  MoveL 4003 to (327.57, -9.53, -317.09) mm, rotated rx -179.9 ry 0 rz -90 deg; joints [33.762, -56.151, 91.428, -130.036, 46.527, 141.521]
  MoveL 4004 to (328.02, -9.53, -316.88) mm, rotated rx -179.9 ry 0 rz -90 deg; joints [33.78, -56.147, 91.421, -130.014, 46.536, 141.505]
  MoveL 4005 to (328.06, -9.53, -316.86) mm, rotated rx -179.9 ry 0 rz -90 deg; joints [33.782, -56.146, 91.42, -130.012, 46.537, 141.503]
  MoveL 4006 to (328.49, -9.53, -316.61) mm, rotated rx -179.9 ry 0 rz -90 deg; joints [33.8, -56.144, 91.417, -129.992, 46.547, 141.489]
  MoveL 4007 to (328.92, -9.53, -316.31) mm, rotated rx -179.9 ry 0 rz -90 deg; joints [33.819, -56.145, 91.417, -129.971, 46.559, 141.475]
  MoveL 4008 to (329.14, -9.53, -316.14) mm, rotated rx -179.9 ry 0 rz -90 deg; joints [33.829, -56.146, 91.419, -129.961, 46.565, 141.468]
  MoveL 4009 to (329.35, -9.52, -315.96) mm, rotated rx -179.9 ry 0 rz -90 deg; joints [33.839, -56.148, 91.422, -129.951, 46.573, 141.462]
  MoveL 4010 to (329.58, -9.52, -315.74) mm, rotated rx -179.9 ry 0 rz -90 deg; joints [33.85, -56.152, 91.427, -129.94, 46.581, 141.456]
  MoveL 4011 to (329.82, -9.52, -315.49) mm, rotated rx -179.9 ry 0 rz -90 deg; joints [33.862, -56.157, 91.435, -129.929, 46.59, 141.45]
  MoveL 4012 to (330, -9.53, -315.27) mm, rotated rx -179.9 ry 0 rz -90 deg; joints [33.872, -56.161, 91.442, -129.92, 46.598, 141.445]
  MoveL 4013 to (330.17, -9.53, -315.06) mm, rotated rx -179.9 ry 0 rz -90 deg; joints [33.882, -56.167, 91.45, -129.912, 46.606, 141.442]
  MoveL 4014 to (330.47, -9.52, -314.63) mm, rotated rx -179.9 ry 0 rz -90 deg; joints [33.9, -56.178, 91.469, -129.898, 46.621, 141.436]
  MoveL 4015 to (330.72, -9.52, -314.2) mm, rotated rx -179.9 ry 0 rz -90 deg; joints [33.916, -56.192, 91.491, -129.886, 46.636, 141.433]
  MoveL 4016 to (330.74, -9.53, -314.16) mm, rotated rx -179.9 ry 0 rz -90 deg; joints [33.917, -56.193, 91.493, -129.885, 46.638, 141.433]
  MoveL 4017 to (330.95, -9.53, -313.71) mm, rotated rx -179.9 ry 0 rz -90 deg; joints [33.933, -56.209, 91.518, -129.876, 46.654, 141.431]
  MoveL 4018 to (331.12, -9.53, -313.26) mm, rotated rx -179.9 ry 0 rz -90 deg; joints [33.947, -56.227, 91.546, -129.868, 46.669, 141.432]
  MoveL 4019 to (331.26, -9.52, -312.81) mm, rotated rx -179.9 ry 0 rz -90 deg; joints [33.96, -56.245, 91.575, -129.862, 46.685, 141.434]
  MoveL 4020 to (331.35, -9.52, -312.37) mm, rotated rx -179.9 ry 0 rz -90 deg; joints [33.972, -56.265, 91.607, -129.857, 46.7, 141.438]
  MoveL 4021 to (331.42, -9.53, -311.92) mm, rotated rx -179.9 ry 0 rz -90 deg; joints [33.983, -56.286, 91.64, -129.854, 46.715, 141.443]
  MoveL 4022 to (331.45, -9.52, -311.47) mm, rotated rx -179.9 ry 0 rz -90 deg; joints [33.993, -56.308, 91.675, -129.853, 46.729, 141.45]
  MoveL 4023 to (331.45, -9.53, -310.57) mm, rotated rx -179.9 ry 0 rz -90 deg; joints [34.012, -56.354, 91.749, -129.853, 46.759, 141.466]
  MoveL 4024 to (331.45, -9.52, -3.46) mm, rotated rx -179.9 ry 0 rz -90 deg; joints [41.448, -70.91, 113.437, -126.774, 55.713, 144.028]
  MoveL 4025 to (331.45, -9.53, -2.56) mm, rotated rx -179.9 ry 0 rz -90 deg; joints [41.474, -70.95, 113.491, -126.757, 55.737, 144.029]
  MoveL 4026 to (331.42, -9.53, -2.11) mm, rotated rx -179.9 ry 0 rz -90 deg; joints [41.486, -70.971, 113.52, -126.75, 55.749, 144.03]
  MoveL 4027 to (331.36, -9.52, -1.67) mm, rotated rx -179.9 ry 0 rz -90 deg; joints [41.497, -70.993, 113.551, -126.744, 55.76, 144.032]
  MoveL 4028 to (331.27, -9.52, -1.22) mm, rotated rx -179.9 ry 0 rz -90 deg; joints [41.506, -71.016, 113.583, -126.739, 55.771, 144.035]
  MoveL 4029 to (331.14, -9.53, -0.77) mm, rotated rx -179.9 ry 0 rz -90 deg; joints [41.515, -71.041, 113.617, -126.735, 55.782, 144.04]
  MoveL 4030 to (330.97, -9.53, -0.32) mm, rotated rx -179.9 ry 0 rz -90 deg; joints [41.523, -71.068, 113.653, -126.733, 55.792, 144.045]
  MoveL 4031 to (330.77, -9.52, 0.13) mm, rotated rx -179.9 ry 0 rz -90 deg; joints [41.529, -71.096, 113.691, -126.733, 55.802, 144.052]
  MoveL 4032 to (330.72, -9.52, 0.23) mm, rotated rx -179.9 ry 0 rz -90 deg; joints [41.53, -71.102, 113.7, -126.733, 55.804, 144.054]
  MoveL 4033 to (330.49, -9.52, 0.63) mm, rotated rx -179.9 ry 0 rz -90 deg; joints [41.534, -71.128, 113.736, -126.735, 55.812, 144.061]
  MoveL 4034 to (330.21, -9.52, 1.03) mm, rotated rx -179.9 ry 0 rz -90 deg; joints [41.537, -71.157, 113.775, -126.738, 55.82, 144.07]
  MoveL 4035 to (330.03, -9.53, 1.27) mm, rotated rx -179.9 ry 0 rz -90 deg; joints [41.538, -71.175, 113.8, -126.74, 55.825, 144.076]
  MoveL 4036 to (329.82, -9.53, 1.51) mm, rotated rx -179.9 ry 0 rz -90 deg; joints [41.538, -71.193, 113.826, -126.744, 55.829, 144.083]
  MoveL 4037 to (329.62, -9.53, 1.72) mm, rotated rx -179.9 ry 0 rz -90 deg; joints [41.537, -71.21, 113.849, -126.748, 55.833, 144.089]
  MoveL 4038 to (329.41, -9.53, 1.93) mm, rotated rx -179.9 ry 0 rz -90 deg; joints [41.536, -71.228, 113.873, -126.752, 55.836, 144.096]
  MoveL 4039 to (329.16, -9.53, 2.14) mm, rotated rx -179.9 ry 0 rz -90 deg; joints [41.535, -71.247, 113.899, -126.758, 55.839, 144.104]
  MoveL 4040 to (328.92, -9.53, 2.33) mm, rotated rx -179.9 ry 0 rz -90 deg; joints [41.532, -71.265, 113.924, -126.764, 55.842, 144.112]
  MoveL 4041 to (328.54, -9.52, 2.6) mm, rotated rx -179.9 ry 0 rz -90 deg; joints [41.528, -71.291, 113.961, -126.774, 55.845, 144.124]
  MoveL 4042 to (328.16, -9.53, 2.82) mm, rotated rx -179.9 ry 0 rz -90 deg; joints [41.522, -71.316, 113.995, -126.785, 55.847, 144.136]
  MoveL 4043 to (328.02, -9.52, 2.9) mm, rotated rx -179.9 ry 0 rz -90 deg; joints [41.519, -71.324, 114.007, -126.789, 55.848, 144.141]
  MoveL 4044 to (327.57, -9.53, 3.11) mm, rotated rx -179.9 ry 0 rz -90 deg; joints [41.511, -71.351, 114.044, -126.803, 55.849, 144.155]
  MoveL 4045 to (327.12, -9.53, 3.28) mm, rotated rx -179.9 ry 0 rz -90 deg; joints [41.501, -71.376, 114.078, -126.817, 55.849, 144.17]
  MoveL 4046 to (326.67, -9.52, 3.41) mm, rotated rx -179.9 ry 0 rz -90 deg; joints [41.491, -71.399, 114.11, -126.833, 55.848, 144.184]
  MoveL 4047 to (326.22, -9.53, 3.51) mm, rotated rx -179.9 ry 0 rz -90 deg; joints [41.479, -71.421, 114.14, -126.849, 55.846, 144.198]
  MoveL 4048 to (325.77, -9.53, 3.57) mm, rotated rx -179.9 ry 0 rz -90 deg; joints [41.466, -71.441, 114.168, -126.866, 55.844, 144.213]
  MoveL 4049 to (325.33, -9.53, 3.6) mm, rotated rx -179.9 ry 0 rz -90 deg; joints [41.452, -71.46, 114.195, -126.883, 55.84, 144.227]
  MoveL 4050 to (324.43, -9.52, 3.61) mm, rotated rx -179.9 ry 0 rz -90 deg; joints [41.423, -71.495, 114.243, -126.919, 55.831, 144.256]
  MoveL 4051 to (319.96, -9.52, 3.61) mm, rotated rx -179.9 ry 0 rz -90 deg; joints [41.278, -71.667, 114.483, -127.098, 55.786, 144.399]
  MoveL 4052 to (319.95, -9.53, 3.61) mm, rotated rx -179.9 ry 0 rz -90 deg; joints [41.278, -71.668, 114.484, -127.098, 55.786, 144.399]
  MoveL 4053 to (319.93, -9.53, 3.62) mm, rotated rx -179.9 ry 0 rz -90 deg; joints [41.277, -71.669, 114.485, -127.099, 55.787, 144.399]
  MoveL 4054 to (319.83, -9.53, 3.72) mm, rotated rx -179.9 ry 0 rz -90 deg; joints [41.277, -71.678, 114.497, -127.101, 55.788, 144.403]
  MoveL 4055 to (319.43, -9.53, 4.05) mm, rotated rx -179.9 ry 0 rz -90 deg; joints [41.273, -71.707, 114.538, -127.11, 55.793, 144.415]
  MoveL 4056 to (319.03, -9.52, 4.33) mm, rotated rx -179.9 ry 0 rz -90 deg; joints [41.268, -71.735, 114.576, -127.121, 55.796, 144.428]
  MoveL 4057 to (318.78, -9.53, 4.48) mm, rotated rx -179.9 ry 0 rz -90 deg; joints [41.265, -71.751, 114.599, -127.128, 55.798, 144.436]
  MoveL 4058 to (318.54, -9.52, 4.62) mm, rotated rx -179.9 ry 0 rz -90 deg; joints [41.26, -71.767, 114.62, -127.135, 55.799, 144.444]
  MoveL 4059 to (318.14, -9.52, 4.81) mm, rotated rx -179.9 ry 0 rz -90 deg; joints [41.253, -71.791, 114.653, -127.147, 55.8, 144.456]
  MoveL 4060 to (317.69, -9.53, 4.99) mm, rotated rx -179.9 ry 0 rz -90 deg; joints [41.243, -71.816, 114.688, -127.162, 55.8, 144.471]
  MoveL 4061 to (317.24, -9.53, 5.13) mm, rotated rx -179.9 ry 0 rz -90 deg; joints [41.233, -71.84, 114.72, -127.177, 55.799, 144.485]
  MoveL 4062 to (316.79, -9.53, 5.23) mm, rotated rx -179.9 ry 0 rz -90 deg; joints [41.221, -71.862, 114.751, -127.193, 55.797, 144.499]
  MoveL 4063 to (316.34, -9.53, 5.3) mm, rotated rx -179.9 ry 0 rz -90 deg; joints [41.208, -71.882, 114.779, -127.21, 55.795, 144.514]
  MoveL 4064 to (315.89, -9.52, 5.34) mm, rotated rx -179.9 ry 0 rz -90 deg; joints [41.195, -71.901, 114.805, -127.227, 55.791, 144.528]
  MoveL 4065 to (315.44, -9.52, 5.35) mm, rotated rx -179.9 ry 0 rz -90 deg; joints [41.18, -71.919, 114.829, -127.245, 55.787, 144.542]
  MoveL 4066 to (-302.86, -9.53, 5.35) mm, rotated rx -179.9 ry 0 rz -90 deg; joints [14.008, -90.074, 136.69, -160.776, 47.297, 167.14]
  MoveL 4067 to (-303.31, -9.52, 5.35) mm, rotated rx -179.9 ry 0 rz -90 deg; joints [13.983, -90.081, 136.697, -160.809, 47.292, 167.161]
  MoveL 4068 to (-303.76, -9.52, 5.31) mm, rotated rx -179.9 ry 0 rz -90 deg; joints [13.958, -90.086, 136.702, -160.842, 47.286, 167.183]
  MoveL 4069 to (-304.21, -9.53, 5.25) mm, rotated rx -179.9 ry 0 rz -90 deg; joints [13.933, -90.089, 136.705, -160.876, 47.281, 167.206]
  MoveL 4070 to (-304.66, -9.53, 5.15) mm, rotated rx -179.9 ry 0 rz -90 deg; joints [13.907, -90.09, 136.706, -160.91, 47.275, 167.229]
  MoveL 4071 to (-305.1, -9.53, 5.01) mm, rotated rx -179.9 ry 0 rz -90 deg; joints [13.881, -90.088, 136.705, -160.945, 47.269, 167.253]
  MoveL 4072 to (-305.55, -9.52, 4.84) mm, rotated rx -179.9 ry 0 rz -90 deg; joints [13.854, -90.084, 136.701, -160.981, 47.264, 167.276]
  MoveL 4073 to (-306.02, -9.52, 4.62) mm, rotated rx -179.9 ry 0 rz -90 deg; joints [13.825, -90.077, 136.695, -161.019, 47.258, 167.302]
  MoveL 4074 to (-306.45, -9.53, 4.37) mm, rotated rx -179.9 ry 0 rz -90 deg; joints [13.798, -90.067, 136.685, -161.055, 47.252, 167.326]
  MoveL 4075 to (-306.88, -9.53, 4.07) mm, rotated rx -179.9 ry 0 rz -90 deg; joints [13.771, -90.054, 136.673, -161.092, 47.247, 167.35]
  MoveL 4076 to (-307.31, -9.52, 3.72) mm, rotated rx -179.9 ry 0 rz -90 deg; joints [13.743, -90.038, 136.657, -161.129, 47.241, 167.376]
  MoveL 4077 to (-307.35, -9.53, 3.68) mm, rotated rx -179.9 ry 0 rz -90 deg; joints [13.74, -90.036, 136.656, -161.133, 47.241, 167.378]
  MoveL 4078 to (-307.41, -9.53, 3.63) mm, rotated rx -179.9 ry 0 rz -90 deg; joints [13.736, -90.033, 136.653, -161.138, 47.24, 167.382]
  MoveL 4079 to (-307.42, -9.53, 3.62) mm, rotated rx -179.9 ry 0 rz -90 deg; joints [13.735, -90.033, 136.652, -161.139, 47.24, 167.382]
  MoveL 4080 to (-307.44, -9.53, 3.61) mm, rotated rx -179.9 ry 0 rz -90 deg; joints [13.734, -90.032, 136.652, -161.141, 47.239, 167.383]
  MoveL 4081 to (-319.03, -9.53, 3.61) mm, rotated rx -179.9 ry 0 rz -90 deg; joints [13.099, -90.213, 136.836, -161.987, 47.104, 167.949]
  MoveL 4082 to (-319.93, -9.52, 3.6) mm, rotated rx -179.9 ry 0 rz -90 deg; joints [13.049, -90.226, 136.849, -162.053, 47.094, 167.993]
  MoveL 4083 to (-320.38, -9.52, 3.56) mm, rotated rx -179.9 ry 0 rz -90 deg; joints [13.024, -90.23, 136.854, -162.087, 47.089, 168.016]
  MoveL 4084 to (-320.83, -9.52, 3.48) mm, rotated rx -179.9 ry 0 rz -90 deg; joints [12.998, -90.232, 136.856, -162.121, 47.084, 168.039]
  MoveL 4085 to (-321.28, -9.53, 3.38) mm, rotated rx -179.9 ry 0 rz -90 deg; joints [12.972, -90.232, 136.856, -162.156, 47.079, 168.062]
  MoveL 4086 to (-321.73, -9.53, 3.24) mm, rotated rx -179.9 ry 0 rz -90 deg; joints [12.946, -90.229, 136.854, -162.192, 47.073, 168.086]
  MoveL 4087 to (-321.8, -9.53, 3.21) mm, rotated rx -179.9 ry 0 rz -90 deg; joints [12.941, -90.229, 136.853, -162.197, 47.072, 168.09]
  MoveC 4088 to (-322.89, -9.52, 3.37) mm, rotated rx -179.9 ry 0 rz -90 deg; joints [12.883, -90.256, 136.88, -162.275, 47.06, 168.142] to (-323.45, -9.52, 4.32) mm, rotated rx -179.9 ry 0 rz -90 deg; joints [12.865, -90.327, 136.95, -162.299, 47.055, 168.158]
  MoveL 4089 to (-323.45, -9.52, 4.32) mm, rotated rx -179.9 ry 0 rz -90 deg; joints [12.865, -90.327, 136.95, -162.299, 47.055, 168.158]
  MoveL 4090 to (-323.82, -9.52, 8.63) mm, rotated rx -179.9 ry 0 rz -90 deg; joints [12.899, -90.621, 137.235, -162.25, 47.054, 168.123]
  MoveL 4091 to (-323.89, -9.15, 9.52) mm, rotated rx -179.9 ry 0 rz -90 deg; joints [12.907, -90.7, 137.28, -162.231, 47.022, 168.103]
  MoveL 4092 to (-323.92, -8.26, 9.89) mm, rotated rx -179.9 ry 0 rz -90 deg; joints [12.909, -90.77, 137.271, -162.205, 46.948, 168.067]
  Set speed (1000.0 mm/s)
  MoveL 4093 to (-323.92, 25.52, 9.89) mm, rotated rx -179.9 ry 0 rz -90 deg; joints [12.895, -92.363, 135.971, -161.337, 44.198, 166.814]
  Print: /'90 deg cut'
  Call SetTool(1)
  Set speed (1000.0 mm/s)
  MoveL 4094 to (-315.62, 25.53, -1.4) mm, rotated rx -179.9 ry 0 rz -90 deg; joints [13.207, -91.468, 135.125, -160.92, 44.317, 166.531]
  MoveL 4095 to (-315.62, 12.75, -1.4) mm, rotated rx -179.9 ry 0 rz -90 deg; joints [13.212, -90.888, 135.622, -161.264, 45.337, 167.021]
  Set speed (100.0 mm/s)
  MoveL 4096 to (-315.62, 5.79, -1.4) mm, rotated rx -179.9 ry 0 rz -90 deg; joints [13.215, -90.564, 135.888, -161.444, 45.896, 167.282]
  MoveC 4097 to (-315.25, 4.9, -1.4) mm, rotated rx -179.9 ry 0 rz -90 deg; joints [13.235, -90.516, 135.916, -161.44, 45.973, 167.296] to (-314.35, 4.53, -1.4) mm, rotated rx -179.9 ry 0 rz -90 deg; joints [13.284, -90.484, 135.916, -161.383, 46.014, 167.265]
  MoveL 4098 to (-314.35, 4.53, -1.4) mm, rotated rx -179.9 ry 0 rz -90 deg; joints [13.284, -90.484, 135.916, -161.383, 46.014, 167.265]
  MoveL 4099 to (-310.68, 4.52, -1.4) mm, rotated rx -179.9 ry 0 rz -90 deg; joints [13.485, -90.427, 135.858, -161.112, 46.058, 167.08]
  MoveC 4100 to (-309.78, 4.52, -1.77) mm, rotated rx -179.9 ry 0 rz -90 deg; joints [13.529, -90.388, 135.819, -161.052, 46.069, 167.04] to (-309.41, 4.53, -2.67) mm, rotated rx -179.9 ry 0 rz -90 deg; joints [13.537, -90.322, 135.755, -161.042, 46.072, 167.033]
  MoveL 4101 to (-309.41, 4.53, -2.67) mm, rotated rx -179.9 ry 0 rz -90 deg; joints [13.537, -90.322, 135.755, -161.042, 46.072, 167.033]
  MoveL 4102 to (-309.41, 4.52, -311.19) mm, rotated rx -179.9 ry 0 rz -90 deg; joints [10.394, -71.426, 113.61, -164.457, 42.297, 168.759]
  MoveL 4103 to (-309.41, 4.53, -311.26) mm, rotated rx -179.9 ry 0 rz -90 deg; joints [10.393, -71.421, 113.604, -164.458, 42.296, 168.759]
  MoveL 4104 to (-309.41, 4.52, -311.3) mm, rotated rx -179.9 ry 0 rz -90 deg; joints [10.393, -71.419, 113.601, -164.458, 42.295, 168.759]
  MoveL 4105 to (-309.41, 4.52, -311.32) mm, rotated rx -179.9 ry 0 rz -90 deg; joints [10.393, -71.418, 113.6, -164.458, 42.295, 168.759]
  MoveC 4106 to (-309.88, 4.52, -312.32) mm, rotated rx -179.9 ry 0 rz -90 deg; joints [10.365, -71.365, 113.527, -164.493, 42.271, 168.781] to (-310.96, 4.53, -312.57) mm, rotated rx -179.9 ry 0 rz -90 deg; joints [10.317, -71.361, 113.523, -164.562, 42.261, 168.831]
  MoveL 4107 to (-310.96, 4.52, -312.57) mm, rotated rx -179.9 ry 0 rz -90 deg; joints [10.317, -71.361, 113.523, -164.562, 42.261, 168.831]
  MoveL 4108 to (-314.37, 4.53, -311.79) mm, rotated rx -179.9 ry 0 rz -90 deg; joints [10.178, -71.442, 113.635, -164.774, 42.263, 168.991]
  MoveL 4109 to (-315.24, 4.9, -311.59) mm, rotated rx -179.9 ry 0 rz -90 deg; joints [10.143, -71.476, 113.652, -164.821, 42.24, 169.022]
  MoveL 4110 to (-315.61, 5.79, -311.51) mm, rotated rx -179.9 ry 0 rz -90 deg; joints [10.128, -71.517, 113.635, -164.826, 42.182, 169.016]
  Set speed (1000.0 mm/s)
  MoveL 4111 to (-315.61, 15.52, -311.51) mm, rotated rx -179.9 ry 0 rz -90 deg; joints [10.125, -71.863, 113.325, -164.637, 41.548, 168.76]
  MoveL 4112 to (-316.42, 15.53, -1.4) mm, rotated rx -179.9 ry 0 rz -90 deg; joints [13.167, -91.028, 135.528, -161.25, 45.105, 166.957]
  MoveL 4113 to (-316.42, 7, -1.4) mm, rotated rx -179.9 ry 0 rz -90 deg; joints [13.171, -90.632, 135.854, -161.472, 45.79, 167.277]
  Set speed (100.0 mm/s)
  MoveL 4114 to (-316.42, 1.27, -1.4) mm, rotated rx -179.9 ry 0 rz -90 deg; joints [13.173, -90.362, 136.07, -161.618, 46.252, 167.489]
  MoveC 4115 to (-316.05, 0.37, -1.4) mm, rotated rx -179.9 ry 0 rz -90 deg; joints [13.194, -90.313, 136.098, -161.613, 46.329, 167.504] to (-315.15, 0, -1.4) mm, rotated rx -179.9 ry 0 rz -90 deg; joints [13.243, -90.282, 136.098, -161.556, 46.369, 167.472]
  MoveL 4116 to (-315.15, 0, -1.4) mm, rotated rx -179.9 ry 0 rz -90 deg; joints [13.243, -90.282, 136.098, -161.556, 46.369, 167.472]
  MoveL 4117 to (-310.68, 0, -1.4) mm, rotated rx -179.9 ry 0 rz -90 deg; joints [13.487, -90.212, 136.028, -161.228, 46.423, 167.25]
  MoveC 4118 to (-309.78, 0, -1.77) mm, rotated rx -179.9 ry 0 rz -90 deg; joints [13.531, -90.173, 135.989, -161.169, 46.433, 167.21] to (-309.41, 0, -2.67) mm, rotated rx -179.9 ry 0 rz -90 deg; joints [13.539, -90.108, 135.925, -161.158, 46.436, 167.203]
  MoveL 4119 to (-309.41, 0, -2.67) mm, rotated rx -179.9 ry 0 rz -90 deg; joints [13.539, -90.108, 135.925, -161.158, 46.436, 167.203]
  MoveL 4120 to (-309.41, 0, -311.19) mm, rotated rx -179.9 ry 0 rz -90 deg; joints [10.395, -71.262, 113.751, -164.544, 42.592, 168.878]
  MoveL 4121 to (-309.41, 0, -311.26) mm, rotated rx -179.9 ry 0 rz -90 deg; joints [10.395, -71.258, 113.745, -164.545, 42.59, 168.878]
  MoveL 4122 to (-309.41, 0, -311.3) mm, rotated rx -179.9 ry 0 rz -90 deg; joints [10.394, -71.255, 113.742, -164.545, 42.589, 168.878]
  MoveL 4123 to (-309.41, 0, -311.32) mm, rotated rx -179.9 ry 0 rz -90 deg; joints [10.394, -71.254, 113.741, -164.545, 42.589, 168.878]
  MoveC 4124 to (-309.88, 0, -312.31) mm, rotated rx -179.9 ry 0 rz -90 deg; joints [10.367, -71.201, 113.669, -164.579, 42.565, 168.899] to (-310.95, 0, -312.57) mm, rotated rx -179.9 ry 0 rz -90 deg; joints [10.319, -71.197, 113.664, -164.648, 42.555, 168.949]
  MoveL 4125 to (-310.95, 0, -312.57) mm, rotated rx -179.9 ry 0 rz -90 deg; joints [10.319, -71.197, 113.664, -164.648, 42.555, 168.949]
  MoveL 4126 to (-315.17, 0, -311.67) mm, rotated rx -179.9 ry 0 rz -90 deg; joints [10.146, -71.294, 113.798, -164.909, 42.558, 169.145]
  MoveL 4127 to (-316.05, 0.37, -311.48) mm, rotated rx -179.9 ry 0 rz -90 deg; joints [10.11, -71.327, 113.814, -164.957, 42.534, 169.176]
  MoveL 4128 to (-316.41, 1.27, -311.4) mm, rotated rx -179.9 ry 0 rz -90 deg; joints [10.095, -71.368, 113.797, -164.962, 42.476, 169.17]
  Set speed (1000.0 mm/s)
  MoveL 4129 to (-316.41, 16.53, -311.4) mm, rotated rx -179.9 ry 0 rz -90 deg; joints [10.091, -71.913, 113.313, -164.669, 41.481, 168.772]
  MoveL 4130 to (328.05, 16.53, -312.66) mm, rotated rx -179.9 ry 0 rz -90 deg; joints [33.855, -57.084, 90.962, -128.897, 45.696, 139.954]
  MoveL 4131 to (328.05, 12.76, -312.66) mm, rotated rx -179.9 ry 0 rz -90 deg; joints [33.857, -56.983, 91.082, -129.063, 45.837, 140.193]
  Set speed (100.0 mm/s)
  MoveL 4132 to (328.05, 5.79, -312.66) mm, rotated rx -179.9 ry 0 rz -90 deg; joints [33.86, -56.792, 91.301, -129.366, 46.098, 140.632]
  MoveL 4133 to (327.68, 4.9, -312.65) mm, rotated rx -179.9 ry 0 rz -90 deg; joints [33.849, -56.781, 91.35, -129.423, 46.129, 140.705]
  MoveL 4134 to (326.78, 4.53, -312.64) mm, rotated rx -179.9 ry 0 rz -90 deg; joints [33.823, -56.802, 91.413, -129.482, 46.139, 140.769]
  MoveL 4135 to (323.18, 4.53, -312.6) mm, rotated rx -179.9 ry 0 rz -90 deg; joints [33.714, -56.928, 91.617, -129.656, 46.12, 140.931]
  MoveC 4136 to (322.29, 4.52, -312.22) mm, rotated rx -179.9 ry 0 rz -90 deg; joints [33.695, -56.978, 91.698, -129.7, 46.127, 140.978] to (321.93, 4.52, -311.32) mm, rotated rx -179.9 ry 0 rz -90 deg; joints [33.702, -57.038, 91.793, -129.718, 46.154, 141.011]
  MoveL 4137 to (321.93, 4.52, -311.32) mm, rotated rx -179.9 ry 0 rz -90 deg; joints [33.702, -57.038, 91.793, -129.718, 46.154, 141.011]
  MoveL 4138 to (321.93, 4.52, -311.3) mm, rotated rx -179.9 ry 0 rz -90 deg; joints [33.703, -57.039, 91.794, -129.718, 46.155, 141.011]
  MoveL 4139 to (321.93, 4.53, -311.26) mm, rotated rx -179.9 ry 0 rz -90 deg; joints [33.703, -57.041, 91.797, -129.718, 46.156, 141.012]
  MoveL 4140 to (321.93, 4.53, -311.04) mm, rotated rx -179.9 ry 0 rz -90 deg; joints [33.708, -57.052, 91.815, -129.718, 46.163, 141.015]
  MoveL 4141 to (321.93, 4.52, -2.67) mm, rotated rx -179.9 ry 0 rz -90 deg; joints [41.154, -71.823, 113.563, -126.625, 55.068, 143.42]
  MoveC 4142 to (322.41, 4.53, -1.67) mm, rotated rx -179.9 ry 0 rz -90 deg; joints [41.198, -71.849, 113.597, -126.587, 55.099, 143.404] to (323.5, 4.53, -1.43) mm, rotated rx -179.9 ry 0 rz -90 deg; joints [41.24, -71.818, 113.553, -126.539, 55.117, 143.369]
  MoveL 4143 to (323.5, 4.52, -1.43) mm, rotated rx -179.9 ry 0 rz -90 deg; joints [41.24, -71.818, 113.553, -126.539, 55.117, 143.369]
  MoveL 4144 to (326.89, 4.53, -2.25) mm, rotated rx -179.9 ry 0 rz -90 deg; joints [41.327, -71.649, 113.322, -126.419, 55.131, 143.26]
  MoveL 4145 to (327.76, 4.9, -2.46) mm, rotated rx -179.9 ry 0 rz -90 deg; joints [41.349, -71.619, 113.25, -126.374, 55.12, 143.207]
  MoveL 4146 to (328.13, 5.8, -2.54) mm, rotated rx -179.9 ry 0 rz -90 deg; joints [41.358, -71.633, 113.197, -126.328, 55.086, 143.137]
  Set speed (1000.0 mm/s)
  MoveL 4147 to (328.13, 15.52, -2.54) mm, rotated rx -179.9 ry 0 rz -90 deg; joints [41.352, -71.977, 112.885, -125.962, 54.696, 142.493]
  MoveL 4148 to (328.88, 15.52, -312.67) mm, rotated rx -179.9 ry 0 rz -90 deg; joints [33.881, -57.028, 90.947, -128.901, 45.738, 139.98]
  MoveL 4149 to (328.88, 7, -312.67) mm, rotated rx -179.9 ry 0 rz -90 deg; joints [33.884, -56.796, 91.216, -129.274, 46.057, 140.519]
  Set speed (100.0 mm/s)
  MoveL 4150 to (328.88, 1.27, -312.67) mm, rotated rx -179.9 ry 0 rz -90 deg; joints [33.887, -56.638, 91.394, -129.52, 46.272, 140.877]
  MoveL 4151 to (328.51, 0.37, -312.66) mm, rotated rx -179.9 ry 0 rz -90 deg; joints [33.876, -56.626, 91.442, -129.577, 46.303, 140.95]
  MoveL 4152 to (327.61, 0, -312.65) mm, rotated rx -179.9 ry 0 rz -90 deg; joints [33.849, -56.647, 91.505, -129.636, 46.313, 141.013]
  MoveL 4153 to (323.18, 0, -312.6) mm, rotated rx -179.9 ry 0 rz -90 deg; joints [33.716, -56.802, 91.756, -129.85, 46.291, 141.213]
  MoveC 4154 to (322.29, 0, -312.22) mm, rotated rx -179.9 ry 0 rz -90 deg; joints [33.697, -56.852, 91.838, -129.893, 46.298, 141.259] to (321.93, 0, -311.32) mm, rotated rx -179.9 ry 0 rz -90 deg; joints [33.704, -56.911, 91.932, -129.911, 46.326, 141.292]
  MoveL 4155 to (321.93, 0, -311.32) mm, rotated rx -179.9 ry 0 rz -90 deg; joints [33.704, -56.911, 91.932, -129.911, 46.326, 141.292]
  MoveL 4156 to (321.93, 0, -311.3) mm, rotated rx -179.9 ry 0 rz -90 deg; joints [33.705, -56.912, 91.934, -129.911, 46.326, 141.292]
  MoveL 4157 to (321.93, 0, -311.26) mm, rotated rx -179.9 ry 0 rz -90 deg; joints [33.705, -56.914, 91.937, -129.911, 46.328, 141.293]
  MoveL 4158 to (321.93, 0, -311.04) mm, rotated rx -179.9 ry 0 rz -90 deg; joints [33.71, -56.926, 91.955, -129.911, 46.335, 141.296]
  MoveL 4159 to (321.93, 0, -2.67) mm, rotated rx -179.9 ry 0 rz -90 deg; joints [41.157, -71.66, 113.705, -126.793, 55.252, 143.716]
  MoveC 4160 to (322.41, 0, -1.67) mm, rotated rx -179.9 ry 0 rz -90 deg; joints [41.201, -71.686, 113.739, -126.755, 55.283, 143.701] to (323.48, 0, -1.43) mm, rotated rx -179.9 ry 0 rz -90 deg; joints [41.243, -71.656, 113.697, -126.707, 55.3, 143.666]
  MoveL 4161 to (323.48, 0, -1.43) mm, rotated rx -179.9 ry 0 rz -90 deg; joints [41.243, -71.656, 113.697, -126.707, 55.3, 143.666]
  MoveL 4162 to (327.69, 0, -2.38) mm, rotated rx -179.9 ry 0 rz -90 deg; joints [41.352, -71.45, 113.412, -126.557, 55.319, 143.531]
  MoveL 4163 to (328.57, 0.37, -2.58) mm, rotated rx -179.9 ry 0 rz -90 deg; joints [41.375, -71.42, 113.341, -126.512, 55.308, 143.478]
  MoveL 4164 to (328.93, 1.27, -2.66) mm, rotated rx -179.9 ry 0 rz -90 deg; joints [41.383, -71.435, 113.289, -126.466, 55.273, 143.407]
  Set speed (1000.0 mm/s)
  MoveL 4165 to (328.93, 25.52, -2.66) mm, rotated rx -179.9 ry 0 rz -90 deg; joints [41.369, -72.285, 112.507, -125.548, 54.305, 141.799]
  Print: /'diagnonal cut'
  Call SetTool(1)
  Set speed (1000.0 mm/s)
  MoveL 4166 to (-336.73, -13.8, 1.64) mm, rotated rx -179.15 ry 0 rz -30.08 deg; joints [-4.609, -80.567, 143.565, -185.552, 62.915, 242.65]
  MoveL 4167 to (-334.14, -15.3, 1.64) mm, rotated rx -179.15 ry 0 rz -30.08 deg; joints [-4.459, -80.469, 143.61, -185.378, 63.051, 242.56]
  Set speed (100.0 mm/s)
  MoveL 4168 to (-328.11, -18.79, 1.64) mm, rotated rx -179.15 ry 0 rz -30.08 deg; joints [-4.111, -80.238, 143.712, -184.973, 63.369, 242.351]
  MoveL 4169 to (-327.17, -18.95, 1.47) mm, rotated rx -179.15 ry 0 rz -30.08 deg; joints [-4.056, -80.22, 143.708, -184.91, 63.38, 242.323]
  MoveL 4170 to (-326.45, -18.45, 1.07) mm, rotated rx -179.15 ry 0 rz -30.08 deg; joints [-4.013, -80.238, 143.672, -184.864, 63.326, 242.306]
  MoveL 4171 to (-325.38, -16.61, 0) mm, rotated rx -179.15 ry 0 rz -30.08 deg; joints [-3.947, -80.317, 143.564, -184.799, 63.137, 242.291]
  MoveC 4172 to (-325.07, -16.06, -0.74) mm, rotated rx -179.15 ry 0 rz -30.08 deg; joints [-3.926, -80.317, 143.502, -184.778, 63.074, 242.286] to (-325.1, -16.12, -1.71) mm, rotated rx -179.15 ry 0 rz -30.08 deg; joints [-3.925, -80.257, 143.435, -184.777, 63.066, 242.286]
  MoveL 4173 to (-325.1, -16.12, -1.71) mm, rotated rx -179.15 ry 0 rz -30.08 deg; joints [-3.925, -80.257, 143.435, -184.777, 63.066, 242.286]
  MoveL 4174 to (-325.19, -16.27, -2.08) mm, rotated rx -179.15 ry 0 rz -30.08 deg; joints [-3.928, -80.225, 143.41, -184.78, 63.074, 242.287]
  MoveL 4175 to (-325.26, -16.39, -2.46) mm, rotated rx -179.15 ry 0 rz -30.08 deg; joints [-3.931, -80.194, 143.386, -184.783, 63.08, 242.288]
  MoveL 4176 to (-325.32, -16.51, -2.91) mm, rotated rx -179.15 ry 0 rz -30.08 deg; joints [-3.933, -80.16, 143.356, -184.785, 63.085, 242.289]
  MoveL 4177 to (-325.37, -16.59, -3.36) mm, rotated rx -179.15 ry 0 rz -30.08 deg; joints [-3.934, -80.128, 143.325, -184.786, 63.086, 242.289]
  MoveL 4178 to (-325.4, -16.65, -3.81) mm, rotated rx -179.15 ry 0 rz -30.08 deg; joints [-3.934, -80.099, 143.294, -184.786, 63.085, 242.289]
  MoveL 4179 to (-325.42, -16.68, -4.26) mm, rotated rx -179.15 ry 0 rz -30.08 deg; joints [-3.933, -80.071, 143.263, -184.785, 63.081, 242.289]
  MoveL 4180 to (-325.42, -16.68, -5.16) mm, rotated rx -179.15 ry 0 rz -30.08 deg; joints [-3.93, -80.02, 143.199, -184.782, 63.068, 242.289]
  MoveL 4181 to (-325.42, -16.68, -310.67) mm, rotated rx -179.15 ry 0 rz -30.08 deg; joints [-3.03, -64.015, 119.968, -184.065, 55.829, 242.408]
  MoveL 4182 to (-325.42, -16.67, -311.57) mm, rotated rx -179.15 ry 0 rz -30.08 deg; joints [-3.028, -63.969, 119.894, -184.064, 55.801, 242.409]
  MoveL 4183 to (-325.4, -16.64, -312.02) mm, rotated rx -179.15 ry 0 rz -30.08 deg; joints [-3.026, -63.949, 119.857, -184.063, 55.784, 242.409]
  MoveL 4184 to (-325.36, -16.57, -312.47) mm, rotated rx -179.15 ry 0 rz -30.08 deg; joints [-3.023, -63.929, 119.82, -184.06, 55.766, 242.408]
  MoveL 4185 to (-325.31, -16.48, -312.92) mm, rotated rx -179.15 ry 0 rz -30.08 deg; joints [-3.02, -63.911, 119.782, -184.057, 55.746, 242.408]
  MoveL 4186 to (-325.24, -16.36, -313.37) mm, rotated rx -179.15 ry 0 rz -30.08 deg; joints [-3.016, -63.895, 119.744, -184.053, 55.724, 242.407]
  MoveL 4187 to (-325.17, -16.25, -313.69) mm, rotated rx -179.15 ry 0 rz -30.08 deg; joints [-3.012, -63.884, 119.716, -184.05, 55.707, 242.406]
  MoveL 4188 to (-325.1, -16.12, -314.02) mm, rotated rx -179.15 ry 0 rz -30.08 deg; joints [-3.008, -63.874, 119.688, -184.046, 55.688, 242.405]
  MoveL 4189 to (-325.04, -16.01, -314.27) mm, rotated rx -179.15 ry 0 rz -30.08 deg; joints [-3.005, -63.867, 119.666, -184.043, 55.673, 242.404]
  MoveL 4190 to (-324.9, -15.78, -314.72) mm, rotated rx -179.15 ry 0 rz -30.08 deg; joints [-2.998, -63.857, 119.626, -184.036, 55.644, 242.402]
  MoveL 4191 to (-324.74, -15.5, -315.17) mm, rotated rx -179.15 ry 0 rz -30.08 deg; joints [-2.99, -63.848, 119.585, -184.028, 55.611, 242.399]
  MoveL 4192 to (-324.65, -15.35, -315.38) mm, rotated rx -179.15 ry 0 rz -30.08 deg; joints [-2.986, -63.845, 119.566, -184.023, 55.595, 242.398]
  MoveL 4193 to (-324.48, -15.05, -315.75) mm, rotated rx -179.15 ry 0 rz -30.08 deg; joints [-2.977, -63.842, 119.532, -184.015, 55.563, 242.394]
  MoveL 4194 to (-324.31, -14.75, -316.07) mm, rotated rx -179.15 ry 0 rz -30.08 deg; joints [-2.969, -63.842, 119.502, -184.006, 55.534, 242.391]
  MoveL 4195 to (-324.2, -14.57, -316.24) mm, rotated rx -179.15 ry 0 rz -30.08 deg; joints [-2.964, -63.842, 119.485, -184.001, 55.517, 242.389]
  MoveL 4196 to (-323.97, -14.18, -316.56) mm, rotated rx -179.15 ry 0 rz -30.08 deg; joints [-2.954, -63.846, 119.454, -183.99, 55.481, 242.385]
  MoveL 4197 to (-323.75, -13.79, -316.83) mm, rotated rx -179.15 ry 0 rz -30.08 deg; joints [-2.943, -63.853, 119.427, -183.979, 55.447, 242.381]
  MoveL 4198 to (-323.61, -13.55, -316.96) mm, rotated rx -179.15 ry 0 rz -30.08 deg; joints [-2.937, -63.858, 119.412, -183.972, 55.427, 242.378]
  MoveL 4199 to (-323.45, -13.28, -317.1) mm, rotated rx -179.15 ry 0 rz -30.08 deg; joints [-2.93, -63.865, 119.397, -183.964, 55.405, 242.375]
  MoveL 4200 to (-323.3, -13.01, -317.22) mm, rotated rx -179.15 ry 0 rz -30.08 deg; joints [-2.923, -63.873, 119.383, -183.957, 55.383, 242.372]
  MoveL 4201 to (-323.07, -12.62, -317.36) mm, rotated rx -179.15 ry 0 rz -30.08 deg; joints [-2.912, -63.886, 119.367, -183.946, 55.353, 242.368]
  MoveL 4202 to (-322.85, -12.23, -317.47) mm, rotated rx -179.15 ry 0 rz -30.08 deg; joints [-2.902, -63.901, 119.353, -183.935, 55.324, 242.363]
  MoveL 4203 to (-322.62, -11.84, -317.54) mm, rotated rx -179.15 ry 0 rz -30.08 deg; joints [-2.893, -63.917, 119.342, -183.924, 55.296, 242.359]
  MoveL 4204 to (-322.4, -11.45, -317.58) mm, rotated rx -179.15 ry 0 rz -30.08 deg; joints [-2.883, -63.935, 119.333, -183.914, 55.269, 242.354]
  MoveL 4205 to (-321.94, -10.67, -317.59) mm, rotated rx -179.15 ry 0 rz -30.08 deg; joints [-2.863, -63.975, 119.322, -183.892, 55.218, 242.345]
  MoveL 4206 to (-316.08, -0.56, -317.59) mm, rotated rx -179.15 ry 0 rz -30.08 deg; joints [-2.608, -64.492, 119.177, -183.611, 54.547, 242.219]
  MoveL 4207 to (-315.63, 0.22, -317.58) mm, rotated rx -179.15 ry 0 rz -30.08 deg; joints [-2.588, -64.532, 119.166, -183.589, 54.496, 242.209]
  MoveL 4208 to (-315.41, 0.61, -317.55) mm, rotated rx -179.15 ry 0 rz -30.08 deg; joints [-2.578, -64.553, 119.163, -183.578, 54.471, 242.204]
  MoveL 4209 to (-315.18, 1, -317.48) mm, rotated rx -179.15 ry 0 rz -30.08 deg; joints [-2.569, -64.576, 119.162, -183.567, 54.447, 242.199]
  MoveL 4210 to (-314.96, 1.39, -317.38) mm, rotated rx -179.15 ry 0 rz -30.08 deg; joints [-2.559, -64.601, 119.165, -183.557, 54.424, 242.194]
  MoveL 4211 to (-314.73, 1.78, -317.24) mm, rotated rx -179.15 ry 0 rz -30.08 deg; joints [-2.55, -64.628, 119.17, -183.546, 54.403, 242.189]
  MoveL 4212 to (-314.56, 2.07, -317.12) mm, rotated rx -179.15 ry 0 rz -30.08 deg; joints [-2.542, -64.649, 119.176, -183.538, 54.387, 242.185]
  MoveL 4213 to (-314.39, 2.37, -316.96) mm, rotated rx -179.15 ry 0 rz -30.08 deg; joints [-2.535, -64.672, 119.184, -183.529, 54.372, 242.181]
  MoveL 4214 to (-314.28, 2.56, -316.85) mm, rotated rx -179.15 ry 0 rz -30.08 deg; joints [-2.531, -64.687, 119.19, -183.524, 54.363, 242.178]
  MoveL 4215 to (-314.17, 2.75, -316.73) mm, rotated rx -179.15 ry 0 rz -30.08 deg; joints [-2.526, -64.703, 119.197, -183.519, 54.353, 242.176]
  MoveL 4216 to (-314.05, 2.95, -316.59) mm, rotated rx -179.15 ry 0 rz -30.08 deg; joints [-2.521, -64.72, 119.205, -183.514, 54.344, 242.173]
  MoveL 4217 to (-313.94, 3.14, -316.44) mm, rotated rx -179.15 ry 0 rz -30.08 deg; joints [-2.517, -64.738, 119.214, -183.508, 54.336, 242.17]
  MoveL 4218 to (-313.83, 3.34, -316.28) mm, rotated rx -179.15 ry 0 rz -30.08 deg; joints [-2.512, -64.756, 119.225, -183.503, 54.328, 242.168]
  MoveL 4219 to (-313.7, 3.57, -316.07) mm, rotated rx -179.15 ry 0 rz -30.08 deg; joints [-2.507, -64.779, 119.239, -183.497, 54.319, 242.164]
  MoveL 4220 to (-313.54, 3.84, -315.78) mm, rotated rx -179.15 ry 0 rz -30.08 deg; joints [-2.5, -64.808, 119.258, -183.489, 54.31, 242.161]
  MoveL 4221 to (-313.38, 4.11, -315.44) mm, rotated rx -179.15 ry 0 rz -30.08 deg; joints [-2.494, -64.839, 119.281, -183.482, 54.301, 242.157]
  MoveL 4222 to (-313.26, 4.31, -315.17) mm, rotated rx -179.15 ry 0 rz -30.08 deg; joints [-2.489, -64.863, 119.301, -183.476, 54.296, 242.154]
  MoveL 4223 to (-313.1, 4.59, -314.72) mm, rotated rx -179.15 ry 0 rz -30.08 deg; joints [-2.483, -64.9, 119.333, -183.469, 54.291, 242.15]
  MoveL 4224 to (-312.96, 4.83, -314.27) mm, rotated rx -179.15 ry 0 rz -30.08 deg; joints [-2.478, -64.935, 119.366, -183.463, 54.289, 242.146]
  MoveL 4225 to (-312.93, 4.89, -314.12) mm, rotated rx -179.15 ry 0 rz -30.08 deg; joints [-2.477, -64.946, 119.377, -183.461, 54.289, 242.145]
  MoveL 4226 to (-312.84, 5.05, -313.75) mm, rotated rx -179.15 ry 0 rz -30.08 deg; joints [-2.474, -64.974, 119.405, -183.457, 54.29, 242.143]
  MoveL 4227 to (-312.76, 5.17, -313.37) mm, rotated rx -179.15 ry 0 rz -30.08 deg; joints [-2.471, -65, 119.434, -183.454, 54.292, 242.141]
  MoveL 4228 to (-312.69, 5.3, -312.92) mm, rotated rx -179.15 ry 0 rz -30.08 deg; joints [-2.469, -65.029, 119.469, -183.451, 54.298, 242.139]
  MoveL 4229 to (-312.64, 5.39, -312.47) mm, rotated rx -179.15 ry 0 rz -30.08 deg; joints [-2.467, -65.057, 119.504, -183.449, 54.305, 242.137]
  MoveL 4230 to (-312.6, 5.45, -312.02) mm, rotated rx -179.15 ry 0 rz -30.08 deg; joints [-2.466, -65.083, 119.539, -183.447, 54.314, 242.136]
  MoveL 4231 to (-312.58, 5.49, -311.57) mm, rotated rx -179.15 ry 0 rz -30.08 deg; joints [-2.466, -65.108, 119.576, -183.447, 54.325, 242.135]
  MoveL 4232 to (-312.58, 5.49, -310.67) mm, rotated rx -179.15 ry 0 rz -30.08 deg; joints [-2.468, -65.155, 119.649, -183.447, 54.351, 242.134]
  MoveL 4233 to (-312.58, 5.49, -3.36) mm, rotated rx -179.15 ry 0 rz -30.08 deg; joints [-3.202, -81.764, 142.908, -184.041, 61.013, 242.082]
  MoveL 4234 to (-312.58, 5.49, -2.46) mm, rotated rx -179.15 ry 0 rz -30.08 deg; joints [-3.205, -81.817, 142.972, -184.044, 61.024, 242.083]
  MoveL 4235 to (-312.6, 5.46, -2.01) mm, rotated rx -179.15 ry 0 rz -30.08 deg; joints [-3.207, -81.841, 143.004, -184.047, 61.032, 242.083]
  MoveL 4236 to (-312.63, 5.4, -1.56) mm, rotated rx -179.15 ry 0 rz -30.08 deg; joints [-3.21, -81.863, 143.037, -184.05, 61.043, 242.084]
  MoveL 4237 to (-312.69, 5.31, -1.11) mm, rotated rx -179.15 ry 0 rz -30.08 deg; joints [-3.215, -81.883, 143.071, -184.055, 61.057, 242.086]
  MoveL 4238 to (-312.75, 5.19, -0.66) mm, rotated rx -179.15 ry 0 rz -30.08 deg; joints [-3.22, -81.901, 143.105, -184.06, 61.073, 242.087]
  MoveL 4239 to (-312.83, 5.06, -0.26) mm, rotated rx -179.15 ry 0 rz -30.08 deg; joints [-3.226, -81.915, 143.136, -184.066, 61.091, 242.089]
  MoveL 4240 to (-312.93, 4.89, 0.14) mm, rotated rx -179.15 ry 0 rz -30.08 deg; joints [-3.233, -81.927, 143.168, -184.073, 61.111, 242.091]
  MoveL 4241 to (-312.95, 4.85, 0.24) mm, rotated rx -179.15 ry 0 rz -30.08 deg; joints [-3.234, -81.929, 143.175, -184.075, 61.116, 242.092]
  MoveL 4242 to (-313.08, 4.62, 0.69) mm, rotated rx -179.15 ry 0 rz -30.08 deg; joints [-3.243, -81.939, 143.212, -184.084, 61.143, 242.094]
  MoveL 4243 to (-313.24, 4.35, 1.14) mm, rotated rx -179.15 ry 0 rz -30.08 deg; joints [-3.254, -81.946, 143.249, -184.095, 61.174, 242.098]
  MoveL 4244 to (-313.38, 4.11, 1.46) mm, rotated rx -179.15 ry 0 rz -30.08 deg; joints [-3.263, -81.948, 143.277, -184.104, 61.2, 242.1]
  MoveL 4245 to (-313.52, 3.87, 1.77) mm, rotated rx -179.15 ry 0 rz -30.08 deg; joints [-3.272, -81.947, 143.303, -184.113, 61.227, 242.103]
  MoveL 4246 to (-313.66, 3.62, 2.03) mm, rotated rx -179.15 ry 0 rz -30.08 deg; joints [-3.281, -81.945, 143.327, -184.123, 61.253, 242.106]
  MoveL 4247 to (-313.83, 3.34, 2.3) mm, rotated rx -179.15 ry 0 rz -30.08 deg; joints [-3.291, -81.94, 143.352, -184.133, 61.283, 242.109]
  MoveL 4248 to (-313.94, 3.14, 2.47) mm, rotated rx -179.15 ry 0 rz -30.08 deg; joints [-3.298, -81.935, 143.367, -184.141, 61.304, 242.112]
  MoveL 4249 to (-314.05, 2.95, 2.61) mm, rotated rx -179.15 ry 0 rz -30.08 deg; joints [-3.305, -81.93, 143.382, -184.148, 61.324, 242.114]
  MoveL 4250 to (-314.17, 2.75, 2.75) mm, rotated rx -179.15 ry 0 rz -30.08 deg; joints [-3.312, -81.923, 143.395, -184.155, 61.344, 242.116]
  MoveL 4251 to (-314.28, 2.56, 2.88) mm, rotated rx -179.15 ry 0 rz -30.08 deg; joints [-3.319, -81.916, 143.408, -184.162, 61.364, 242.118]
  MoveL 4252 to (-314.33, 2.46, 2.93) mm, rotated rx -179.15 ry 0 rz -30.08 deg; joints [-3.323, -81.913, 143.414, -184.165, 61.373, 242.119]
  MoveL 4253 to (-314.53, 2.12, 3.11) mm, rotated rx -179.15 ry 0 rz -30.08 deg; joints [-3.335, -81.898, 143.434, -184.178, 61.408, 242.123]
  MoveL 4254 to (-314.73, 1.78, 3.26) mm, rotated rx -179.15 ry 0 rz -30.08 deg; joints [-3.346, -81.882, 143.451, -184.19, 61.442, 242.126]
  MoveL 4255 to (-314.96, 1.39, 3.4) mm, rotated rx -179.15 ry 0 rz -30.08 deg; joints [-3.36, -81.861, 143.468, -184.204, 61.48, 242.13]
  MoveL 4256 to (-315.18, 1, 3.5) mm, rotated rx -179.15 ry 0 rz -30.08 deg; joints [-3.373, -81.838, 143.483, -184.217, 61.518, 242.134]
  MoveL 4257 to (-315.41, 0.61, 3.57) mm, rotated rx -179.15 ry 0 rz -30.08 deg; joints [-3.386, -81.813, 143.496, -184.231, 61.556, 242.138]
  MoveL 4258 to (-315.63, 0.22, 3.6) mm, rotated rx -179.15 ry 0 rz -30.08 deg; joints [-3.399, -81.787, 143.506, -184.244, 61.593, 242.142]
  MoveL 4259 to (-316.08, -0.56, 3.61) mm, rotated rx -179.15 ry 0 rz -30.08 deg; joints [-3.426, -81.729, 143.522, -184.271, 61.667, 242.15]
  MoveL 4260 to (-316.53, -1.33, 3.61) mm, rotated rx -179.15 ry 0 rz -30.08 deg; joints [-3.451, -81.672, 143.537, -184.297, 61.741, 242.158]
  MoveL 4261 to (-316.98, -2.11, 3.58) mm, rotated rx -179.15 ry 0 rz -30.08 deg; joints [-3.477, -81.613, 143.55, -184.324, 61.814, 242.165]
  MoveL 4262 to (-317.44, -2.89, 3.46) mm, rotated rx -179.15 ry 0 rz -30.08 deg; joints [-3.503, -81.547, 143.557, -184.35, 61.887, 242.173]
  MoveL 4263 to (-322.4, -11.45, 1.89) mm, rotated rx -179.15 ry 0 rz -30.08 deg; joints [-3.783, -80.815, 143.607, -184.634, 62.676, 242.25]
  MoveL 4264 to (-322.85, -12.23, 1.75) mm, rotated rx -179.15 ry 0 rz -30.08 deg; joints [-3.808, -80.748, 143.611, -184.659, 62.748, 242.256]
  MoveL 4265 to (-323.07, -12.62, 1.64) mm, rotated rx -179.15 ry 0 rz -30.08 deg; joints [-3.821, -80.713, 143.61, -184.672, 62.783, 242.259]
  MoveL 4266 to (-323.3, -13.01, 1.5) mm, rotated rx -179.15 ry 0 rz -30.08 deg; joints [-3.833, -80.675, 143.607, -184.684, 62.818, 242.263]
  MoveL 4267 to (-323.51, -13.37, 1.34) mm, rotated rx -179.15 ry 0 rz -30.08 deg; joints [-3.845, -80.638, 143.602, -184.696, 62.85, 242.266]
  MoveL 4268 to (-323.72, -13.74, 1.14) mm, rotated rx -179.15 ry 0 rz -30.08 deg; joints [-3.856, -80.6, 143.594, -184.707, 62.882, 242.268]
  MoveL 4269 to (-323.75, -13.79, 1.1) mm, rotated rx -179.15 ry 0 rz -30.08 deg; joints [-3.858, -80.594, 143.593, -184.709, 62.886, 242.269]
  MoveL 4270 to (-323.97, -14.18, 0.84) mm, rotated rx -179.15 ry 0 rz -30.08 deg; joints [-3.87, -80.549, 143.581, -184.721, 62.919, 242.272]
  MoveL 4271 to (-324.2, -14.57, 0.52) mm, rotated rx -179.15 ry 0 rz -30.08 deg; joints [-3.881, -80.501, 143.565, -184.733, 62.951, 242.275]
  MoveL 4272 to (-324.37, -14.86, 0.24) mm, rotated rx -179.15 ry 0 rz -30.08 deg; joints [-3.89, -80.464, 143.55, -184.742, 62.975, 242.277]
  MoveL 4273 to (-324.52, -15.12, -0.05) mm, rotated rx -179.15 ry 0 rz -30.08 deg; joints [-3.897, -80.427, 143.534, -184.749, 62.995, 242.279]
  MoveL 4274 to (-324.65, -15.35, -0.34) mm, rotated rx -179.15 ry 0 rz -30.08 deg; joints [-3.904, -80.394, 143.518, -184.756, 63.013, 242.281]
  MoveL 4275 to (-324.78, -15.57, -0.66) mm, rotated rx -179.15 ry 0 rz -30.08 deg; joints [-3.91, -80.358, 143.499, -184.762, 63.029, 242.282]
  MoveL 4276 to (-324.94, -15.84, -1.11) mm, rotated rx -179.15 ry 0 rz -30.08 deg; joints [-3.917, -80.313, 143.472, -184.769, 63.048, 242.284]
  MoveL 4277 to (-325.06, -16.06, -1.56) mm, rotated rx -179.15 ry 0 rz -30.08 deg; joints [-3.923, -80.27, 143.444, -184.775, 63.062, 242.286]
  MoveL 4278 to (-325.1, -16.12, -1.71) mm, rotated rx -179.15 ry 0 rz -30.08 deg; joints [-3.925, -80.257, 143.435, -184.777, 63.066, 242.286]
  MoveC 4279 to (-325.47, -16.76, -2.34) mm, rotated rx -179.15 ry 0 rz -30.08 deg; joints [-3.943, -80.173, 143.4, -184.795, 63.117, 242.291] to (-325.96, -17.6, -2.27) mm, rotated rx -179.15 ry 0 rz -30.08 deg; joints [-3.971, -80.114, 143.42, -184.824, 63.197, 242.298]
  MoveL 4280 to (-325.96, -17.6, -2.27) mm, rotated rx -179.15 ry 0 rz -30.08 deg; joints [-3.971, -80.114, 143.42, -184.824, 63.197, 242.298]
  MoveC 4281 to (-326.58, -18.68, -2.33) mm, rotated rx -179.15 ry 0 rz -30.08 deg; joints [-4.007, -80.028, 143.434, -184.859, 63.298, 242.306] to (-326.88, -19.19, -3.44) mm, rotated rx -179.15 ry 0 rz -30.08 deg; joints [-4.02, -79.927, 143.365, -184.872, 63.329, 242.309]
  MoveL 4282 to (-326.88, -19.19, -3.44) mm, rotated rx -179.15 ry 0 rz -30.08 deg; joints [-4.02, -79.927, 143.365, -184.872, 63.329, 242.309]
  MoveC 4283 to (-327, -19.4, -4.21) mm, rotated rx -179.15 ry 0 rz -30.08 deg; joints [-4.024, -79.867, 143.313, -184.876, 63.337, 242.311] to (-327.34, -19.98, -4.68) mm, rotated rx -179.15 ry 0 rz -30.08 deg; joints [-4.041, -79.797, 143.289, -184.893, 63.384, 242.315]
  MoveL 4284 to (-327.34, -19.98, -4.68) mm, rotated rx -179.15 ry 0 rz -30.08 deg; joints [-4.041, -79.797, 143.289, -184.893, 63.384, 242.315]
  MoveC 4285 to (-328.33, -21.7, -4.92) mm, rotated rx -179.15 ry 0 rz -30.08 deg; joints [-4.097, -79.654, 143.301, -184.949, 63.541, 242.327] to (-329.31, -23.38, -4.5) mm, rotated rx -179.15 ry 0 rz -30.08 deg; joints [-4.154, -79.549, 143.359, -185.006, 63.705, 242.34]
  MoveL 4286 to (-329.31, -23.38, -4.5) mm, rotated rx -179.15 ry 0 rz -30.08 deg; joints [-4.154, -79.549, 143.359, -185.006, 63.705, 242.34]
  MoveL 4287 to (-329.33, -23.42, -4.48) mm, rotated rx -179.15 ry 0 rz -30.08 deg; joints [-4.155, -79.547, 143.361, -185.007, 63.709, 242.34]
  MoveL 4288 to (-329.99, -24.68, -3.66) mm, rotated rx -179.15 ry 0 rz -30.08 deg; joints [-4.197, -79.497, 143.44, -185.048, 63.84, 242.348]
  MoveL 4289 to (-330.52, -25.7, -2.49) mm, rotated rx -179.15 ry 0 rz -30.08 deg; joints [-4.231, -79.484, 143.541, -185.082, 63.955, 242.354]
  MoveL 4290 to (-330.86, -26.42, -1.05) mm, rotated rx -179.15 ry 0 rz -30.08 deg; joints [-4.257, -79.51, 143.656, -185.106, 64.045, 242.357]
  MoveL 4291 to (-331, -26.79, 0.94) mm, rotated rx -179.15 ry 0 rz -30.08 deg; joints [-4.273, -79.591, 143.804, -185.121, 64.111, 242.358]
  MoveL 4292 to (-330.79, -26.58, 2.94) mm, rotated rx -179.15 ry 0 rz -30.08 deg; joints [-4.27, -79.72, 143.944, -185.117, 64.123, 242.356]
  MoveL 4293 to (-330.27, -25.81, 4.73) mm, rotated rx -179.15 ry 0 rz -30.08 deg; joints [-4.247, -79.88, 144.06, -185.094, 64.078, 242.349]
  MoveL 4294 to (-329.47, -24.58, 6.12) mm, rotated rx -179.15 ry 0 rz -30.08 deg; joints [-4.207, -80.054, 144.139, -185.053, 63.981, 242.339]
  MoveL 4295 to (-328.48, -23.02, 6.95) mm, rotated rx -179.15 ry 0 rz -30.08 deg; joints [-4.154, -80.222, 144.172, -185, 63.845, 242.326]
  MoveL 4296 to (-327.41, -21.31, 7.12) mm, rotated rx -179.15 ry 0 rz -30.08 deg; joints [-4.092, -80.363, 144.155, -184.938, 63.685, 242.312]
  MoveL 4297 to (-326.37, -19.65, 6.61) mm, rotated rx -179.15 ry 0 rz -30.08 deg; joints [-4.03, -80.463, 144.091, -184.876, 63.52, 242.296]
  MoveL 4298 to (-325.52, -18.32, 5.58) mm, rotated rx -179.15 ry 0 rz -30.08 deg; joints [-3.977, -80.507, 143.995, -184.822, 63.378, 242.283]
  MoveL 4299 to (-324.87, -17.33, 4.11) mm, rotated rx -179.15 ry 0 rz -30.08 deg; joints [-3.934, -80.5, 143.874, -184.778, 63.262, 242.272]
  MoveL 4300 to (-324.48, -16.78, 2.35) mm, rotated rx -179.15 ry 0 rz -30.08 deg; joints [-3.904, -80.442, 143.739, -184.749, 63.185, 242.265]
  MoveL 4301 to (-324.37, -16.73, 0.46) mm, rotated rx -179.15 ry 0 rz -30.08 deg; joints [-3.891, -80.339, 143.605, -184.735, 63.153, 242.261]
  MoveL 4302 to (-324.56, -17.19, -1.36) mm, rotated rx -179.15 ry 0 rz -30.08 deg; joints [-3.895, -80.201, 143.483, -184.739, 63.17, 242.261]
  MoveL 4303 to (-325.11, -18.29, -3.15) mm, rotated rx -179.15 ry 0 rz -30.08 deg; joints [-3.919, -80.016, 143.375, -184.763, 63.247, 242.267]
  MoveL 4304 to (-325.94, -19.88, -4.39) mm, rotated rx -179.15 ry 0 rz -30.08 deg; joints [-3.962, -79.827, 143.314, -184.805, 63.377, 242.276]
  MoveL 4305 to (-326.93, -21.74, -4.92) mm, rotated rx -179.15 ry 0 rz -30.08 deg; joints [-4.017, -79.656, 143.309, -184.859, 63.543, 242.287]
  MoveL 4306 to (-327.95, -23.65, -4.66) mm, rotated rx -179.15 ry 0 rz -30.08 deg; joints [-4.076, -79.526, 143.36, -184.918, 63.726, 242.299]
  MoveL 4307 to (-328.85, -25.35, -3.65) mm, rotated rx -179.15 ry 0 rz -30.08 deg; joints [-4.131, -79.452, 143.46, -184.972, 63.902, 242.31]
  MoveL 4308 to (-329.51, -26.64, -2.03) mm, rotated rx -179.15 ry 0 rz -30.08 deg; joints [-4.175, -79.444, 143.598, -185.015, 64.049, 242.317]
  MoveL 4309 to (-329.83, -27.35, 0) mm, rotated rx -179.15 ry 0 rz -30.08 deg; joints [-4.202, -79.503, 143.755, -185.041, 64.147, 242.32]
  MoveL 4310 to (-329.77, -27.39, 2.18) mm, rotated rx -179.15 ry 0 rz -30.08 deg; joints [-4.208, -79.621, 143.911, -185.045, 64.186, 242.319]
  MoveL 4311 to (-329.32, -26.77, 4.21) mm, rotated rx -179.15 ry 0 rz -30.08 deg; joints [-4.19, -79.783, 144.046, -185.027, 64.158, 242.313]
  MoveL 4312 to (-328.53, -25.56, 5.85) mm, rotated rx -179.15 ry 0 rz -30.08 deg; joints [-4.151, -79.968, 144.143, -184.987, 64.068, 242.303]
  MoveL 4313 to (-327.5, -23.94, 6.86) mm, rotated rx -179.15 ry 0 rz -30.08 deg; joints [-4.096, -80.152, 144.189, -184.932, 63.929, 242.29]
  MoveL 4314 to (-326.35, -22.11, 7.13) mm, rotated rx -179.15 ry 0 rz -30.08 deg; joints [-4.031, -80.309, 144.177, -184.866, 63.758, 242.274]
  MoveL 4315 to (-325.23, -20.32, 6.61) mm, rotated rx -179.15 ry 0 rz -30.08 deg; joints [-3.964, -80.418, 144.11, -184.799, 63.58, 242.258]
  MoveL 4316 to (-324.38, -18.98, 5.58) mm, rotated rx -179.15 ry 0 rz -30.08 deg; joints [-3.91, -80.462, 144.014, -184.745, 63.438, 242.244]
  MoveL 4317 to (-323.73, -17.99, 4.11) mm, rotated rx -179.15 ry 0 rz -30.08 deg; joints [-3.867, -80.455, 143.892, -184.702, 63.323, 242.233]
  MoveL 4318 to (-323.33, -17.44, 2.35) mm, rotated rx -179.15 ry 0 rz -30.08 deg; joints [-3.838, -80.397, 143.758, -184.672, 63.246, 242.226]
  MoveL 4319 to (-323.23, -17.39, 0.46) mm, rotated rx -179.15 ry 0 rz -30.08 deg; joints [-3.825, -80.294, 143.623, -184.658, 63.214, 242.222]
  MoveL 4320 to (-323.42, -17.85, -1.36) mm, rotated rx -179.15 ry 0 rz -30.08 deg; joints [-3.829, -80.157, 143.502, -184.662, 63.23, 242.222]
  MoveL 4321 to (-323.92, -18.86, -3.04) mm, rotated rx -179.15 ry 0 rz -30.08 deg; joints [-3.851, -79.986, 143.4, -184.684, 63.3, 242.227]
  MoveL 4322 to (-324.67, -20.29, -4.26) mm, rotated rx -179.15 ry 0 rz -30.08 deg; joints [-3.889, -79.809, 143.338, -184.722, 63.416, 242.236]
  MoveL 4323 to (-325.57, -21.99, -4.87) mm, rotated rx -179.15 ry 0 rz -30.08 deg; joints [-3.938, -79.646, 143.324, -184.771, 63.566, 242.246]
  MoveL 4324 to (-326.52, -23.78, -4.81) mm, rotated rx -179.15 ry 0 rz -30.08 deg; joints [-3.993, -79.514, 143.358, -184.825, 63.734, 242.258]
  MoveL 4325 to (-327.41, -25.45, -4.09) mm, rotated rx -179.15 ry 0 rz -30.08 deg; joints [-4.046, -79.427, 143.438, -184.878, 63.901, 242.268]
  MoveL 4326 to (-328.12, -26.82, -2.79) mm, rotated rx -179.15 ry 0 rz -30.08 deg; joints [-4.092, -79.394, 143.554, -184.923, 64.051, 242.276]
  MoveL 4327 to (-328.57, -27.74, -1.05) mm, rotated rx -179.15 ry 0 rz -30.08 deg; joints [-4.125, -79.42, 143.693, -184.954, 64.165, 242.281]
  MoveL 4328 to (-328.71, -28.12, 0.93) mm, rotated rx -179.15 ry 0 rz -30.08 deg; joints [-4.141, -79.501, 143.841, -184.969, 64.232, 242.282]
  MoveL 4329 to (-328.51, -27.91, 2.92) mm, rotated rx -179.15 ry 0 rz -30.08 deg; joints [-4.138, -79.629, 143.98, -184.965, 64.244, 242.28]
  MoveL 4330 to (-327.98, -27.15, 4.72) mm, rotated rx -179.15 ry 0 rz -30.08 deg; joints [-4.115, -79.788, 144.096, -184.941, 64.2, 242.273]
  MoveL 4331 to (-327.19, -25.92, 6.11) mm, rotated rx -179.15 ry 0 rz -30.08 deg; joints [-4.075, -79.961, 144.175, -184.901, 64.105, 242.263]
  MoveL 4332 to (-326.21, -24.37, 6.94) mm, rotated rx -179.15 ry 0 rz -30.08 deg; joints [-4.021, -80.129, 144.209, -184.847, 63.969, 242.249]
  MoveL 4333 to (-325.14, -22.67, 7.12) mm, rotated rx -179.15 ry 0 rz -30.08 deg; joints [-3.96, -80.271, 144.193, -184.786, 63.81, 242.235]
  MoveL 4334 to (-324.1, -21.01, 6.63) mm, rotated rx -179.15 ry 0 rz -30.08 deg; joints [-3.898, -80.371, 144.131, -184.723, 63.645, 242.219]
  MoveL 4335 to (-324.08, -20.98, 6.61) mm, rotated rx -179.15 ry 0 rz -30.08 deg; joints [-3.897, -80.373, 144.129, -184.722, 63.641, 242.219]
  MoveL 4336 to (-323.77, -20.44, 6.33) mm, rotated rx -179.15 ry 0 rz -30.08 deg; joints [-3.878, -80.399, 144.099, -184.703, 63.586, 242.215]
  MoveC 4337 to (-322.17, -17.67, 2.95) mm, rotated rx -179.15 ry 0 rz -30.08 deg; joints [-3.773, -80.419, 143.811, -184.598, 63.274, 242.19] to (-322.23, -17.79, -1.71) mm, rotated rx -179.15 ry 0 rz -30.08 deg; joints [-3.759, -80.146, 143.481, -184.585, 63.217, 242.189]
  MoveL 4338 to (-322.23, -17.79, -1.71) mm, rotated rx -179.15 ry 0 rz -30.08 deg; joints [-3.759, -80.146, 143.481, -184.585, 63.217, 242.189]
  MoveL 4339 to (-322.32, -17.93, -2.08) mm, rotated rx -179.15 ry 0 rz -30.08 deg; joints [-3.763, -80.114, 143.457, -184.588, 63.225, 242.19]
  MoveL 4340 to (-322.39, -18.05, -2.46) mm, rotated rx -179.15 ry 0 rz -30.08 deg; joints [-3.765, -80.084, 143.432, -184.591, 63.231, 242.19]
  MoveL 4341 to (-322.45, -18.17, -2.91) mm, rotated rx -179.15 ry 0 rz -30.08 deg; joints [-3.767, -80.05, 143.402, -184.593, 63.235, 242.191]
  MoveL 4342 to (-322.5, -18.25, -3.36) mm, rotated rx -179.15 ry 0 rz -30.08 deg; joints [-3.769, -80.018, 143.372, -184.595, 63.237, 242.192]
  MoveL 4343 to (-322.54, -18.31, -3.81) mm, rotated rx -179.15 ry 0 rz -30.08 deg; joints [-3.769, -79.988, 143.341, -184.595, 63.235, 242.192]
  MoveL 4344 to (-322.55, -18.34, -4.26) mm, rotated rx -179.15 ry 0 rz -30.08 deg; joints [-3.768, -79.961, 143.309, -184.594, 63.231, 242.192]
  MoveL 4345 to (-322.55, -18.34, -5.16) mm, rotated rx -179.15 ry 0 rz -30.08 deg; joints [-3.765, -79.91, 143.245, -184.591, 63.218, 242.191]
  MoveL 4346 to (-322.55, -18.34, -310.67) mm, rotated rx -179.15 ry 0 rz -30.08 deg; joints [-2.903, -63.938, 120.005, -183.908, 55.938, 242.313]
  MoveL 4347 to (-322.55, -18.33, -311.57) mm, rotated rx -179.15 ry 0 rz -30.08 deg; joints [-2.901, -63.893, 119.932, -183.906, 55.909, 242.314]
  MoveL 4348 to (-322.53, -18.3, -312.02) mm, rotated rx -179.15 ry 0 rz -30.08 deg; joints [-2.9, -63.872, 119.895, -183.905, 55.893, 242.314]
  MoveL 4349 to (-322.49, -18.24, -312.47) mm, rotated rx -179.15 ry 0 rz -30.08 deg; joints [-2.897, -63.853, 119.857, -183.903, 55.875, 242.314]
  MoveL 4350 to (-322.44, -18.14, -312.92) mm, rotated rx -179.15 ry 0 rz -30.08 deg; joints [-2.894, -63.835, 119.819, -183.9, 55.855, 242.313]
  MoveL 4351 to (-322.37, -18.02, -313.37) mm, rotated rx -179.15 ry 0 rz -30.08 deg; joints [-2.89, -63.818, 119.781, -183.896, 55.833, 242.312]
  MoveL 4352 to (-322.31, -17.91, -313.69) mm, rotated rx -179.15 ry 0 rz -30.08 deg; joints [-2.886, -63.808, 119.753, -183.892, 55.816, 242.311]
  MoveL 4353 to (-322.23, -17.79, -314.02) mm, rotated rx -179.15 ry 0 rz -30.08 deg; joints [-2.882, -63.798, 119.725, -183.888, 55.797, 242.31]
  MoveL 4354 to (-322.17, -17.67, -314.27) mm, rotated rx -179.15 ry 0 rz -30.08 deg; joints [-2.879, -63.791, 119.703, -183.885, 55.782, 242.309]
  MoveL 4355 to (-322.03, -17.44, -314.72) mm, rotated rx -179.15 ry 0 rz -30.08 deg; joints [-2.872, -63.78, 119.663, -183.878, 55.752, 242.307]
  MoveL 4356 to (-321.87, -17.16, -315.17) mm, rotated rx -179.15 ry 0 rz -30.08 deg; joints [-2.864, -63.772, 119.623, -183.87, 55.72, 242.304]
  MoveL 4357 to (-321.78, -17.01, -315.38) mm, rotated rx -179.15 ry 0 rz -30.08 deg; joints [-2.86, -63.769, 119.603, -183.865, 55.703, 242.303]
  MoveL 4358 to (-321.61, -16.71, -315.75) mm, rotated rx -179.15 ry 0 rz -30.08 deg; joints [-2.851, -63.766, 119.569, -183.857, 55.672, 242.299]
  MoveL 4359 to (-321.44, -16.41, -316.07) mm, rotated rx -179.15 ry 0 rz -30.08 deg; joints [-2.843, -63.766, 119.539, -183.848, 55.642, 242.296]
  MoveL 4360 to (-321.33, -16.23, -316.24) mm, rotated rx -179.15 ry 0 rz -30.08 deg; joints [-2.838, -63.766, 119.523, -183.843, 55.625, 242.294]
  MoveL 4361 to (-321.11, -15.84, -316.56) mm, rotated rx -179.15 ry 0 rz -30.08 deg; joints [-2.828, -63.77, 119.491, -183.832, 55.589, 242.29]
  MoveL 4362 to (-320.88, -15.45, -316.83) mm, rotated rx -179.15 ry 0 rz -30.08 deg; joints [-2.817, -63.777, 119.464, -183.821, 55.555, 242.286]
  MoveL 4363 to (-320.74, -15.22, -316.96) mm, rotated rx -179.15 ry 0 rz -30.08 deg; joints [-2.811, -63.782, 119.45, -183.814, 55.535, 242.283]
  MoveL 4364 to (-320.59, -14.94, -317.1) mm, rotated rx -179.15 ry 0 rz -30.08 deg; joints [-2.804, -63.789, 119.434, -183.807, 55.513, 242.28]
  MoveL 4365 to (-320.43, -14.67, -317.22) mm, rotated rx -179.15 ry 0 rz -30.08 deg; joints [-2.797, -63.797, 119.421, -183.799, 55.491, 242.277]
  MoveL 4366 to (-320.2, -14.28, -317.36) mm, rotated rx -179.15 ry 0 rz -30.08 deg; joints [-2.787, -63.81, 119.404, -183.788, 55.461, 242.272]
  MoveL 4367 to (-319.98, -13.89, -317.47) mm, rotated rx -179.15 ry 0 rz -30.08 deg; joints [-2.777, -63.825, 119.39, -183.777, 55.432, 242.268]
  MoveL 4368 to (-319.75, -13.5, -317.54) mm, rotated rx -179.15 ry 0 rz -30.08 deg; joints [-2.767, -63.841, 119.379, -183.766, 55.405, 242.263]
  MoveL 4369 to (-319.53, -13.12, -317.58) mm, rotated rx -179.15 ry 0 rz -30.08 deg; joints [-2.757, -63.859, 119.371, -183.756, 55.378, 242.258]
  MoveL 4370 to (-319.08, -12.34, -317.59) mm, rotated rx -179.15 ry 0 rz -30.08 deg; joints [-2.737, -63.899, 119.36, -183.734, 55.326, 242.249]
  MoveL 4371 to (-312.31, -0.66, -317.59) mm, rotated rx -179.15 ry 0 rz -30.08 deg; joints [-2.443, -64.495, 119.192, -183.408, 54.553, 242.102]
  MoveL 4372 to (-311.86, 0.12, -317.58) mm, rotated rx -179.15 ry 0 rz -30.08 deg; joints [-2.423, -64.535, 119.18, -183.386, 54.501, 242.091]
  MoveL 4373 to (-311.64, 0.51, -317.56) mm, rotated rx -179.15 ry 0 rz -30.08 deg; joints [-2.413, -64.556, 119.176, -183.375, 54.476, 242.086]
  MoveL 4374 to (-311.41, 0.9, -317.5) mm, rotated rx -179.15 ry 0 rz -30.08 deg; joints [-2.404, -64.579, 119.175, -183.364, 54.452, 242.081]
  MoveL 4375 to (-311.19, 1.29, -317.41) mm, rotated rx -179.15 ry 0 rz -30.08 deg; joints [-2.394, -64.603, 119.177, -183.353, 54.429, 242.076]
  MoveL 4376 to (-310.96, 1.67, -317.28) mm, rotated rx -179.15 ry 0 rz -30.08 deg; joints [-2.385, -64.629, 119.181, -183.342, 54.407, 242.071]
  MoveL 4377 to (-310.76, 2.02, -317.14) mm, rotated rx -179.15 ry 0 rz -30.08 deg; joints [-2.376, -64.654, 119.187, -183.333, 54.388, 242.066]
  MoveL 4378 to (-310.56, 2.37, -316.96) mm, rotated rx -179.15 ry 0 rz -30.08 deg; joints [-2.368, -64.681, 119.196, -183.323, 54.37, 242.061]
  MoveL 4379 to (-310.51, 2.45, -316.92) mm, rotated rx -179.15 ry 0 rz -30.08 deg; joints [-2.366, -64.687, 119.199, -183.321, 54.366, 242.06]
  MoveL 4380 to (-310.28, 2.84, -316.67) mm, rotated rx -179.15 ry 0 rz -30.08 deg; joints [-2.356, -64.72, 119.213, -183.31, 54.347, 242.055]
  MoveL 4381 to (-310.17, 3.04, -316.53) mm, rotated rx -179.15 ry 0 rz -30.08 deg; joints [-2.351, -64.737, 119.222, -183.305, 54.339, 242.052]
  MoveL 4382 to (-310.06, 3.23, -316.37) mm, rotated rx -179.15 ry 0 rz -30.08 deg; joints [-2.347, -64.755, 119.232, -183.299, 54.33, 242.049]
  MoveL 4383 to (-309.86, 3.57, -316.07) mm, rotated rx -179.15 ry 0 rz -30.08 deg; joints [-2.339, -64.787, 119.251, -183.29, 54.317, 242.044]
  MoveL 4384 to (-309.74, 3.79, -315.83) mm, rotated rx -179.15 ry 0 rz -30.08 deg; joints [-2.334, -64.811, 119.267, -183.284, 54.309, 242.041]
  MoveL 4385 to (-309.61, 4.01, -315.58) mm, rotated rx -179.15 ry 0 rz -30.08 deg; joints [-2.329, -64.835, 119.284, -183.278, 54.302, 242.038]
  MoveL 4386 to (-309.43, 4.31, -315.17) mm, rotated rx -179.15 ry 0 rz -30.08 deg; joints [-2.322, -64.872, 119.313, -183.269, 54.294, 242.033]
  MoveL 4387 to (-309.28, 4.57, -314.76) mm, rotated rx -179.15 ry 0 rz -30.08 deg; joints [-2.316, -64.906, 119.342, -183.263, 54.289, 242.03]
  MoveL 4388 to (-309.16, 4.79, -314.35) mm, rotated rx -179.15 ry 0 rz -30.08 deg; joints [-2.311, -64.938, 119.372, -183.257, 54.287, 242.026]
  MoveL 4389 to (-309.13, 4.83, -314.27) mm, rotated rx -179.15 ry 0 rz -30.08 deg; joints [-2.31, -64.944, 119.378, -183.256, 54.287, 242.026]
  MoveL 4390 to (-309.02, 5.02, -313.82) mm, rotated rx -179.15 ry 0 rz -30.08 deg; joints [-2.306, -64.977, 119.412, -183.251, 54.287, 242.023]
  MoveL 4391 to (-308.93, 5.17, -313.37) mm, rotated rx -179.15 ry 0 rz -30.08 deg; joints [-2.303, -65.008, 119.446, -183.247, 54.29, 242.02]
  MoveL 4392 to (-308.86, 5.3, -312.92) mm, rotated rx -179.15 ry 0 rz -30.08 deg; joints [-2.3, -65.038, 119.481, -183.244, 54.296, 242.018]
  MoveL 4393 to (-308.81, 5.39, -312.47) mm, rotated rx -179.15 ry 0 rz -30.08 deg; joints [-2.299, -65.065, 119.516, -183.241, 54.303, 242.017]
  MoveL 4394 to (-308.77, 5.45, -312.02) mm, rotated rx -179.15 ry 0 rz -30.08 deg; joints [-2.298, -65.092, 119.552, -183.24, 54.312, 242.015]
  MoveL 4395 to (-308.75, 5.49, -311.57) mm, rotated rx -179.15 ry 0 rz -30.08 deg; joints [-2.298, -65.117, 119.588, -183.239, 54.323, 242.015]
  MoveL 4396 to (-308.75, 5.49, -310.67) mm, rotated rx -179.15 ry 0 rz -30.08 deg; joints [-2.299, -65.164, 119.661, -183.24, 54.349, 242.014]
  MoveL 4397 to (-308.75, 5.49, -3.36) mm, rotated rx -179.15 ry 0 rz -30.08 deg; joints [-2.981, -81.777, 142.922, -183.789, 61.007, 241.961]
  MoveL 4398 to (-308.75, 5.49, -2.46) mm, rotated rx -179.15 ry 0 rz -30.08 deg; joints [-2.984, -81.829, 142.986, -183.792, 61.018, 241.961]
  MoveL 4399 to (-308.77, 5.46, -2.01) mm, rotated rx -179.15 ry 0 rz -30.08 deg; joints [-2.986, -81.854, 143.018, -183.795, 61.026, 241.962]
  MoveL 4400 to (-308.8, 5.4, -1.56) mm, rotated rx -179.15 ry 0 rz -30.08 deg; joints [-2.99, -81.876, 143.051, -183.798, 61.037, 241.963]
  MoveL 4401 to (-308.85, 5.31, -1.11) mm, rotated rx -179.15 ry 0 rz -30.08 deg; joints [-2.994, -81.896, 143.085, -183.802, 61.051, 241.964]
  MoveL 4402 to (-308.92, 5.19, -0.66) mm, rotated rx -179.15 ry 0 rz -30.08 deg; joints [-2.999, -81.914, 143.119, -183.808, 61.067, 241.966]
  MoveL 4403 to (-309.01, 5.04, -0.21) mm, rotated rx -179.15 ry 0 rz -30.08 deg; joints [-3.005, -81.929, 143.154, -183.814, 61.087, 241.968]
  MoveL 4404 to (-309.12, 4.85, 0.24) mm, rotated rx -179.15 ry 0 rz -30.08 deg; joints [-3.013, -81.942, 143.189, -183.822, 61.11, 241.97]
  MoveL 4405 to (-309.16, 4.79, 0.37) mm, rotated rx -179.15 ry 0 rz -30.08 deg; joints [-3.015, -81.945, 143.2, -183.825, 61.117, 241.971]
  MoveL 4406 to (-309.27, 4.59, 0.75) mm, rotated rx -179.15 ry 0 rz -30.08 deg; joints [-3.023, -81.953, 143.231, -183.833, 61.141, 241.974]
  MoveL 4407 to (-309.41, 4.35, 1.14) mm, rotated rx -179.15 ry 0 rz -30.08 deg; joints [-3.032, -81.958, 143.263, -183.842, 61.168, 241.977]
  MoveL 4408 to (-309.5, 4.19, 1.37) mm, rotated rx -179.15 ry 0 rz -30.08 deg; joints [-3.038, -81.96, 143.283, -183.848, 61.186, 241.979]
  MoveL 4409 to (-309.61, 4.01, 1.6) mm, rotated rx -179.15 ry 0 rz -30.08 deg; joints [-3.045, -81.961, 143.303, -183.855, 61.205, 241.981]
  MoveL 4410 to (-309.72, 3.81, 1.83) mm, rotated rx -179.15 ry 0 rz -30.08 deg; joints [-3.052, -81.96, 143.323, -183.863, 61.226, 241.983]
  MoveL 4411 to (-309.83, 3.62, 2.03) mm, rotated rx -179.15 ry 0 rz -30.08 deg; joints [-3.059, -81.958, 143.341, -183.87, 61.247, 241.985]
  MoveL 4412 to (-309.95, 3.43, 2.22) mm, rotated rx -179.15 ry 0 rz -30.08 deg; joints [-3.066, -81.955, 143.359, -183.877, 61.268, 241.988]
  MoveL 4413 to (-310.06, 3.23, 2.39) mm, rotated rx -179.15 ry 0 rz -30.08 deg; joints [-3.073, -81.95, 143.375, -183.884, 61.288, 241.99]
  MoveL 4414 to (-310.17, 3.04, 2.55) mm, rotated rx -179.15 ry 0 rz -30.08 deg; joints [-3.08, -81.945, 143.389, -183.892, 61.308, 241.992]
  MoveL 4415 to (-310.28, 2.85, 2.69) mm, rotated rx -179.15 ry 0 rz -30.08 deg; joints [-3.087, -81.94, 143.403, -183.899, 61.328, 241.994]
  MoveL 4416 to (-310.5, 2.46, 2.93) mm, rotated rx -179.15 ry 0 rz -30.08 deg; joints [-3.101, -81.926, 143.428, -183.913, 61.367, 241.999]
  MoveL 4417 to (-310.51, 2.45, 2.94) mm, rotated rx -179.15 ry 0 rz -30.08 deg; joints [-3.101, -81.925, 143.429, -183.913, 61.368, 241.999]
  MoveL 4418 to (-310.73, 2.06, 3.14) mm, rotated rx -179.15 ry 0 rz -30.08 deg; joints [-3.115, -81.909, 143.451, -183.927, 61.408, 242.003]
  MoveL 4419 to (-310.96, 1.67, 3.3) mm, rotated rx -179.15 ry 0 rz -30.08 deg; joints [-3.128, -81.89, 143.471, -183.941, 61.446, 242.007]
  MoveL 4420 to (-311.19, 1.29, 3.43) mm, rotated rx -179.15 ry 0 rz -30.08 deg; joints [-3.142, -81.868, 143.487, -183.955, 61.485, 242.012]
  MoveL 4421 to (-311.41, 0.9, 3.52) mm, rotated rx -179.15 ry 0 rz -30.08 deg; joints [-3.155, -81.845, 143.502, -183.968, 61.523, 242.016]
  MoveL 4422 to (-311.64, 0.51, 3.58) mm, rotated rx -179.15 ry 0 rz -30.08 deg; joints [-3.168, -81.82, 143.513, -183.982, 61.56, 242.02]
  MoveL 4423 to (-311.86, 0.12, 3.6) mm, rotated rx -179.15 ry 0 rz -30.08 deg; joints [-3.181, -81.792, 143.523, -183.996, 61.597, 242.024]
  MoveL 4424 to (-312.31, -0.66, 3.61) mm, rotated rx -179.15 ry 0 rz -30.08 deg; joints [-3.207, -81.735, 143.539, -184.022, 61.671, 242.032]
  MoveL 4425 to (-313.67, -3, 3.61) mm, rotated rx -179.15 ry 0 rz -30.08 deg; joints [-3.285, -81.562, 143.585, -184.102, 61.892, 242.056]
  MoveL 4426 to (-314.12, -3.77, 3.58) mm, rotated rx -179.15 ry 0 rz -30.08 deg; joints [-3.311, -81.503, 143.598, -184.129, 61.966, 242.064]
  MoveL 4427 to (-314.57, -4.55, 3.46) mm, rotated rx -179.15 ry 0 rz -30.08 deg; joints [-3.337, -81.437, 143.605, -184.155, 62.038, 242.072]
  MoveL 4428 to (-319.53, -13.12, 1.89) mm, rotated rx -179.15 ry 0 rz -30.08 deg; joints [-3.617, -80.704, 143.654, -184.441, 62.828, 242.151]
  MoveL 4429 to (-319.98, -13.89, 1.75) mm, rotated rx -179.15 ry 0 rz -30.08 deg; joints [-3.642, -80.637, 143.658, -184.466, 62.9, 242.157]
  MoveL 4430 to (-320.2, -14.28, 1.64) mm, rotated rx -179.15 ry 0 rz -30.08 deg; joints [-3.655, -80.602, 143.657, -184.479, 62.935, 242.161]
  MoveL 4431 to (-320.43, -14.67, 1.5) mm, rotated rx -179.15 ry 0 rz -30.08 deg; joints [-3.667, -80.564, 143.654, -184.492, 62.97, 242.164]
  MoveL 4432 to (-320.64, -15.04, 1.34) mm, rotated rx -179.15 ry 0 rz -30.08 deg; joints [-3.679, -80.527, 143.649, -184.503, 63.002, 242.167]
  MoveL 4433 to (-320.85, -15.4, 1.14) mm, rotated rx -179.15 ry 0 rz -30.08 deg; joints [-3.69, -80.489, 143.641, -184.515, 63.033, 242.17]
  MoveL 4434 to (-320.88, -15.45, 1.1) mm, rotated rx -179.15 ry 0 rz -30.08 deg; joints [-3.692, -80.483, 143.64, -184.516, 63.038, 242.171]
  MoveL 4435 to (-321.11, -15.84, 0.84) mm, rotated rx -179.15 ry 0 rz -30.08 deg; joints [-3.704, -80.438, 143.628, -184.529, 63.071, 242.174]
  MoveL 4436 to (-321.33, -16.23, 0.52) mm, rotated rx -179.15 ry 0 rz -30.08 deg; joints [-3.716, -80.39, 143.612, -184.541, 63.103, 242.177]
  MoveL 4437 to (-321.5, -16.52, 0.24) mm, rotated rx -179.15 ry 0 rz -30.08 deg; joints [-3.724, -80.353, 143.597, -184.549, 63.126, 242.179]
  MoveL 4438 to (-321.65, -16.78, -0.05) mm, rotated rx -179.15 ry 0 rz -30.08 deg; joints [-3.732, -80.317, 143.581, -184.557, 63.146, 242.181]
  MoveL 4439 to (-321.78, -17.01, -0.34) mm, rotated rx -179.15 ry 0 rz -30.08 deg; joints [-3.738, -80.283, 143.565, -184.564, 63.164, 242.183]
  MoveL 4440 to (-321.91, -17.23, -0.66) mm, rotated rx -179.15 ry 0 rz -30.08 deg; joints [-3.745, -80.248, 143.546, -184.57, 63.18, 242.185]
  MoveL 4441 to (-322.07, -17.5, -1.11) mm, rotated rx -179.15 ry 0 rz -30.08 deg; joints [-3.752, -80.202, 143.519, -184.577, 63.199, 242.187]
  MoveL 4442 to (-322.2, -17.72, -1.56) mm, rotated rx -179.15 ry 0 rz -30.08 deg; joints [-3.758, -80.159, 143.491, -184.583, 63.213, 242.188]
  MoveL 4443 to (-322.23, -17.79, -1.71) mm, rotated rx -179.15 ry 0 rz -30.08 deg; joints [-3.759, -80.146, 143.481, -184.585, 63.217, 242.189]
  MoveC 4444 to (-322.67, -18.54, -2.38) mm, rotated rx -179.15 ry 0 rz -30.08 deg; joints [-3.782, -80.051, 143.447, -184.608, 63.278, 242.195] to (-323.21, -19.47, -2.12) mm, rotated rx -179.15 ry 0 rz -30.08 deg; joints [-3.813, -79.996, 143.481, -184.639, 63.369, 242.202]
  MoveL 4445 to (-323.21, -19.47, -2.12) mm, rotated rx -179.15 ry 0 rz -30.08 deg; joints [-3.813, -79.996, 143.481, -184.639, 63.369, 242.202]
  MoveL 4446 to (-324.81, -22.23, 0.52) mm, rotated rx -179.15 ry 0 rz -30.08 deg; joints [-3.915, -79.933, 143.717, -184.741, 63.669, 242.225]
  MoveL 4447 to (-325.48, -22.64, 1.09) mm, rotated rx -179.15 ry 0 rz -30.08 deg; joints [-3.956, -79.932, 143.762, -184.785, 63.718, 242.241]
  MoveL 4448 to (-326.4, -22.44, 1.33) mm, rotated rx -179.15 ry 0 rz -30.08 deg; joints [-4.01, -79.957, 143.771, -184.846, 63.704, 242.269]
  Set speed (1000.0 mm/s)
  MoveL 4449 to (-337.88, -15.79, 1.33) mm, rotated rx -179.15 ry 0 rz -30.08 deg; joints [-4.673, -80.398, 143.577, -185.616, 63.099, 242.663]
  Print: /'Parallel1'
  Call SetTool(1)
  Set speed (1000.0 mm/s)
  MoveL 4450 to (-338.94, 18.29, -0.93) mm, rotated rx -179.15 ry 0 rz -30.08 deg; joints [-4.729, -82.692, 142.659, -185.853, 59.905, 243.058]
  MoveL 4451 to (-318.25, 6.3, -0.93) mm, rotated rx -179.15 ry 0 rz -30.08 deg; joints [-3.536, -81.944, 143.039, -184.426, 60.976, 242.27]
  Set speed (100.0 mm/s)
  MoveL 4452 to (-317.62, 5.94, -0.93) mm, rotated rx -179.15 ry 0 rz -30.08 deg; joints [-3.5, -81.921, 143.05, -184.383, 61.009, 242.247]
  MoveC 4453 to (-317.03, 5.16, -0.93) mm, rotated rx -179.15 ry 0 rz -30.08 deg; joints [-3.466, -81.868, 143.07, -184.341, 61.08, 242.222] to (-317.15, 4.2, -0.93) mm, rotated rx -179.15 ry 0 rz -30.08 deg; joints [-3.473, -81.799, 143.091, -184.345, 61.17, 242.218]
  MoveL 4454 to (-317.15, 4.2, -0.93) mm, rotated rx -179.15 ry 0 rz -30.08 deg; joints [-3.473, -81.799, 143.091, -184.345, 61.17, 242.218]
  MoveL 4455 to (-326.56, -12.05, -0.93) mm, rotated rx -179.15 ry 0 rz -30.08 deg; joints [-4.012, -80.594, 143.399, -184.891, 62.699, 242.366]
  MoveC 4456 to (-326.65, -12.16, -0.93) mm, rotated rx -179.15 ry 0 rz -30.08 deg; joints [-4.017, -80.585, 143.401, -184.896, 62.71, 242.368] to (-326.76, -12.26, -0.93) mm, rotated rx -179.15 ry 0 rz -30.08 deg; joints [-4.024, -80.578, 143.403, -184.903, 62.719, 242.37]
  MoveL 4457 to (-326.76, -12.26, -0.93) mm, rotated rx -179.15 ry 0 rz -30.08 deg; joints [-4.024, -80.578, 143.403, -184.903, 62.719, 242.37]
  MoveC 4458 to (-326.87, -12.35, -0.93) mm, rotated rx -179.15 ry 0 rz -30.08 deg; joints [-4.03, -80.57, 143.404, -184.91, 62.728, 242.372] to (-326.96, -12.46, -0.93) mm, rotated rx -179.15 ry 0 rz -30.08 deg; joints [-4.035, -80.561, 143.406, -184.915, 62.739, 242.374]
  MoveL 4459 to (-326.96, -12.46, -0.93) mm, rotated rx -179.15 ry 0 rz -30.08 deg; joints [-4.035, -80.561, 143.406, -184.915, 62.739, 242.374]
  MoveL 4460 to (-327.56, -13.5, -0.93) mm, rotated rx -179.15 ry 0 rz -30.08 deg; joints [-4.069, -80.483, 143.424, -184.949, 62.836, 242.382]
  MoveC 4461 to (-328.23, -14.66, -1.49) mm, rotated rx -179.15 ry 0 rz -30.08 deg; joints [-4.106, -80.364, 143.405, -184.986, 62.938, 242.391] to (-328.51, -15.15, -2.84) mm, rotated rx -179.15 ry 0 rz -30.08 deg; joints [-4.116, -80.251, 143.318, -184.996, 62.964, 242.394]
  MoveL 4462 to (-328.51, -15.15, -2.84) mm, rotated rx -179.15 ry 0 rz -30.08 deg; joints [-4.116, -80.251, 143.318, -184.996, 62.964, 242.394]
  MoveL 4463 to (-328.51, -15.15, -5.37) mm, rotated rx -179.15 ry 0 rz -30.08 deg; joints [-4.106, -80.107, 143.137, -184.987, 62.927, 242.392]
  MoveC 4464 to (-328.23, -14.66, -6.72) mm, rotated rx -179.15 ry 0 rz -30.08 deg; joints [-4.085, -80.067, 143.033, -184.966, 62.862, 242.388] to (-327.56, -13.5, -7.28) mm, rotated rx -179.15 ry 0 rz -30.08 deg; joints [-4.044, -80.123, 142.972, -184.925, 62.744, 242.378]
  MoveL 4465 to (-327.56, -13.5, -7.28) mm, rotated rx -179.15 ry 0 rz -30.08 deg; joints [-4.044, -80.123, 142.972, -184.925, 62.744, 242.378]
  MoveC 4466 to (-327.47, -13.38, -7.28) mm, rotated rx -179.15 ry 0 rz -30.08 deg; joints [-4.039, -80.131, 142.97, -184.92, 62.734, 242.377] to (-327.36, -13.29, -7.28) mm, rotated rx -179.15 ry 0 rz -30.08 deg; joints [-4.033, -80.139, 142.969, -184.913, 62.725, 242.374]
  MoveL 4467 to (-327.36, -13.29, -7.28) mm, rotated rx -179.15 ry 0 rz -30.08 deg; joints [-4.033, -80.139, 142.969, -184.913, 62.725, 242.374]
  MoveL 4468 to (-327.36, -13.29, -7.28) mm, rotated rx -179.15 ry 0 rz -30.08 deg; joints [-4.033, -80.139, 142.969, -184.913, 62.725, 242.374]
  MoveC 4469 to (-327.25, -13.2, -7.28) mm, rotated rx -179.15 ry 0 rz -30.08 deg; joints [-4.027, -80.146, 142.968, -184.907, 62.716, 242.372] to (-327.16, -13.08, -7.28) mm, rotated rx -179.15 ry 0 rz -30.08 deg; joints [-4.022, -80.154, 142.966, -184.901, 62.705, 242.37]
  MoveL 4470 to (-327.16, -13.08, -7.28) mm, rotated rx -179.15 ry 0 rz -30.08 deg; joints [-4.022, -80.154, 142.966, -184.901, 62.705, 242.37]
  MoveL 4471 to (-316.67, 5.04, -7.28) mm, rotated rx -179.15 ry 0 rz -30.08 deg; joints [-3.424, -81.488, 142.625, -184.296, 61.014, 242.205]
  MoveC 4472 to (-316.61, 5.17, -7.28) mm, rotated rx -179.15 ry 0 rz -30.08 deg; joints [-3.42, -81.497, 142.622, -184.292, 61.002, 242.204] to (-316.59, 5.31, -7.28) mm, rotated rx -179.15 ry 0 rz -30.08 deg; joints [-3.419, -81.507, 142.619, -184.291, 60.988, 242.204]
  MoveL 4473 to (-316.59, 5.31, -7.28) mm, rotated rx -179.15 ry 0 rz -30.08 deg; joints [-3.419, -81.507, 142.619, -184.291, 60.988, 242.204]
  MoveC 4474 to (-316.56, 5.45, -7.28) mm, rotated rx -179.15 ry 0 rz -30.08 deg; joints [-3.417, -81.517, 142.616, -184.29, 60.975, 242.205] to (-316.5, 5.58, -7.28) mm, rotated rx -179.15 ry 0 rz -30.08 deg; joints [-3.414, -81.527, 142.613, -184.287, 60.963, 242.204]
  MoveL 4475 to (-316.5, 5.58, -7.28) mm, rotated rx -179.15 ry 0 rz -30.08 deg; joints [-3.414, -81.527, 142.613, -184.287, 60.963, 242.204]
  MoveL 4476 to (-316.49, 5.6, -7.28) mm, rotated rx -179.15 ry 0 rz -30.08 deg; joints [-3.414, -81.528, 142.613, -184.286, 60.961, 242.204]
  MoveC 4477 to (-315.82, 6.77, -7.84) mm, rotated rx -179.15 ry 0 rz -30.08 deg; joints [-3.373, -81.579, 142.55, -184.245, 60.846, 242.191] to (-315.54, 7.25, -9.18) mm, rotated rx -179.15 ry 0 rz -30.08 deg; joints [-3.353, -81.535, 142.445, -184.224, 60.784, 242.185]
  MoveL 4478 to (-315.54, 7.25, -9.18) mm, rotated rx -179.15 ry 0 rz -30.08 deg; joints [-3.353, -81.535, 142.445, -184.224, 60.784, 242.185]
  MoveL 4479 to (-315.54, 7.25, -11.72) mm, rotated rx -179.15 ry 0 rz -30.08 deg; joints [-3.345, -81.386, 142.265, -184.216, 60.753, 242.183]
  MoveC 4480 to (-315.82, 6.77, -13.07) mm, rotated rx -179.15 ry 0 rz -30.08 deg; joints [-3.356, -81.273, 142.179, -184.228, 60.781, 242.187] to (-316.49, 5.6, -13.63) mm, rotated rx -179.15 ry 0 rz -30.08 deg; joints [-3.393, -81.157, 142.163, -184.265, 60.882, 242.199]
  MoveL 4481 to (-316.49, 5.6, -13.63) mm, rotated rx -179.15 ry 0 rz -30.08 deg; joints [-3.393, -81.157, 142.163, -184.265, 60.882, 242.199]
  MoveC 4482 to (-316.55, 5.47, -13.63) mm, rotated rx -179.15 ry 0 rz -30.08 deg; joints [-3.396, -81.148, 142.165, -184.269, 60.894, 242.2] to (-316.58, 5.33, -13.63) mm, rotated rx -179.15 ry 0 rz -30.08 deg; joints [-3.397, -81.138, 142.168, -184.27, 60.907, 242.199]
  MoveL 4483 to (-316.58, 5.33, -13.63) mm, rotated rx -179.15 ry 0 rz -30.08 deg; joints [-3.397, -81.138, 142.168, -184.27, 60.907, 242.199]
  MoveC 4484 to (-316.6, 5.18, -13.63) mm, rotated rx -179.15 ry 0 rz -30.08 deg; joints [-3.399, -81.128, 142.171, -184.271, 60.92, 242.199] to (-316.66, 5.05, -13.63) mm, rotated rx -179.15 ry 0 rz -30.08 deg; joints [-3.402, -81.118, 142.174, -184.274, 60.932, 242.2]
  MoveL 4485 to (-316.66, 5.05, -13.63) mm, rotated rx -179.15 ry 0 rz -30.08 deg; joints [-3.402, -81.118, 142.174, -184.274, 60.932, 242.2]
  MoveL 4486 to (-327.16, -13.08, -13.63) mm, rotated rx -179.15 ry 0 rz -30.08 deg; joints [-3.997, -79.795, 142.513, -184.878, 62.611, 242.367]
  MoveC 4487 to (-327.25, -13.2, -13.63) mm, rotated rx -179.15 ry 0 rz -30.08 deg; joints [-4.002, -79.787, 142.515, -184.883, 62.622, 242.368] to (-327.36, -13.29, -13.63) mm, rotated rx -179.15 ry 0 rz -30.08 deg; joints [-4.008, -79.779, 142.516, -184.889, 62.63, 242.37]
  MoveL 4488 to (-327.36, -13.29, -13.63) mm, rotated rx -179.15 ry 0 rz -30.08 deg; joints [-4.008, -79.779, 142.516, -184.889, 62.63, 242.37]
  MoveC 4489 to (-327.47, -13.38, -13.63) mm, rotated rx -179.15 ry 0 rz -30.08 deg; joints [-4.014, -79.772, 142.517, -184.896, 62.639, 242.373] to (-327.56, -13.5, -13.63) mm, rotated rx -179.15 ry 0 rz -30.08 deg; joints [-4.019, -79.764, 142.519, -184.901, 62.65, 242.374]
  MoveL 4490 to (-327.56, -13.5, -13.63) mm, rotated rx -179.15 ry 0 rz -30.08 deg; joints [-4.019, -79.764, 142.519, -184.901, 62.65, 242.374]
  MoveC 4491 to (-328.23, -14.66, -14.19) mm, rotated rx -179.15 ry 0 rz -30.08 deg; joints [-4.055, -79.646, 142.5, -184.937, 62.749, 242.383] to (-328.51, -15.15, -15.53) mm, rotated rx -179.15 ry 0 rz -30.08 deg; joints [-4.066, -79.534, 142.412, -184.948, 62.773, 242.386]
  MoveL 4492 to (-328.51, -15.15, -15.53) mm, rotated rx -179.15 ry 0 rz -30.08 deg; joints [-4.066, -79.534, 142.412, -184.948, 62.773, 242.386]
  MoveL 4493 to (-328.51, -15.15, -18.07) mm, rotated rx -179.15 ry 0 rz -30.08 deg; joints [-4.056, -79.392, 142.23, -184.939, 62.733, 242.385]
  MoveC 4494 to (-328.23, -14.66, -19.42) mm, rotated rx -179.15 ry 0 rz -30.08 deg; joints [-4.035, -79.352, 142.125, -184.918, 62.668, 242.381] to (-327.56, -13.5, -19.98) mm, rotated rx -179.15 ry 0 rz -30.08 deg; joints [-3.995, -79.406, 142.065, -184.878, 62.552, 242.371]
  MoveL 4495 to (-327.56, -13.5, -19.98) mm, rotated rx -179.15 ry 0 rz -30.08 deg; joints [-3.995, -79.406, 142.065, -184.878, 62.552, 242.371]
  MoveL 4496 to (-327.55, -13.5, -19.98) mm, rotated rx -179.15 ry 0 rz -30.08 deg; joints [-3.994, -79.407, 142.065, -184.878, 62.552, 242.371]
  MoveC 4497 to (-327.47, -13.38, -19.98) mm, rotated rx -179.15 ry 0 rz -30.08 deg; joints [-3.99, -79.415, 142.063, -184.873, 62.541, 242.369] to (-327.36, -13.29, -19.98) mm, rotated rx -179.15 ry 0 rz -30.08 deg; joints [-3.983, -79.422, 142.062, -184.866, 62.533, 242.367]
  MoveL 4498 to (-327.36, -13.29, -19.98) mm, rotated rx -179.15 ry 0 rz -30.08 deg; joints [-3.983, -79.422, 142.062, -184.866, 62.533, 242.367]
  MoveC 4499 to (-327.25, -13.19, -19.98) mm, rotated rx -179.15 ry 0 rz -30.08 deg; joints [-3.977, -79.429, 142.06, -184.859, 62.524, 242.365] to (-327.16, -13.08, -19.98) mm, rotated rx -179.15 ry 0 rz -30.08 deg; joints [-3.972, -79.438, 142.059, -184.854, 62.513, 242.363]
  MoveL 4500 to (-327.16, -13.08, -19.98) mm, rotated rx -179.15 ry 0 rz -30.08 deg; joints [-3.972, -79.438, 142.059, -184.854, 62.513, 242.363]
  MoveL 4501 to (-316.66, 5.05, -19.98) mm, rotated rx -179.15 ry 0 rz -30.08 deg; joints [-3.381, -80.75, 141.722, -184.254, 60.849, 242.195]
  MoveC 4502 to (-316.6, 5.19, -19.98) mm, rotated rx -179.15 ry 0 rz -30.08 deg; joints [-3.378, -80.759, 141.72, -184.251, 60.837, 242.195] to (-316.58, 5.33, -19.98) mm, rotated rx -179.15 ry 0 rz -30.08 deg; joints [-3.377, -80.769, 141.717, -184.25, 60.824, 242.195]
  MoveL 4503 to (-316.58, 5.33, -19.98) mm, rotated rx -179.15 ry 0 rz -30.08 deg; joints [-3.377, -80.769, 141.717, -184.25, 60.824, 242.195]
  MoveC 4504 to (-316.55, 5.47, -19.98) mm, rotated rx -179.15 ry 0 rz -30.08 deg; joints [-3.375, -80.779, 141.714, -184.248, 60.811, 242.195] to (-316.49, 5.6, -19.98) mm, rotated rx -179.15 ry 0 rz -30.08 deg; joints [-3.372, -80.788, 141.711, -184.245, 60.799, 242.194]
  MoveL 4505 to (-316.49, 5.6, -19.98) mm, rotated rx -179.15 ry 0 rz -30.08 deg; joints [-3.372, -80.788, 141.711, -184.245, 60.799, 242.194]
  MoveC 4506 to (-315.82, 6.77, -20.53) mm, rotated rx -179.15 ry 0 rz -30.08 deg; joints [-3.332, -80.838, 141.648, -184.204, 60.684, 242.182] to (-315.54, 7.25, -21.88) mm, rotated rx -179.15 ry 0 rz -30.08 deg; joints [-3.312, -80.794, 141.543, -184.184, 60.622, 242.176]
  MoveL 4507 to (-315.54, 7.25, -21.88) mm, rotated rx -179.15 ry 0 rz -30.08 deg; joints [-3.312, -80.794, 141.543, -184.184, 60.622, 242.176]
  MoveL 4508 to (-315.54, 7.25, -24.42) mm, rotated rx -179.15 ry 0 rz -30.08 deg; joints [-3.304, -80.647, 141.362, -184.176, 60.588, 242.174]
  MoveC 4509 to (-315.82, 6.77, -25.77) mm, rotated rx -179.15 ry 0 rz -30.08 deg; joints [-3.316, -80.535, 141.275, -184.188, 60.614, 242.178] to (-316.49, 5.6, -26.33) mm, rotated rx -179.15 ry 0 rz -30.08 deg; joints [-3.352, -80.421, 141.258, -184.225, 60.712, 242.19]
  MoveL 4510 to (-316.49, 5.6, -26.33) mm, rotated rx -179.15 ry 0 rz -30.08 deg; joints [-3.352, -80.421, 141.258, -184.225, 60.712, 242.19]
  MoveC 4511 to (-316.55, 5.47, -26.33) mm, rotated rx -179.15 ry 0 rz -30.08 deg; joints [-3.355, -80.412, 141.261, -184.229, 60.724, 242.191] to (-316.58, 5.33, -26.33) mm, rotated rx -179.15 ry 0 rz -30.08 deg; joints [-3.356, -80.402, 141.264, -184.23, 60.737, 242.191]
  MoveL 4512 to (-316.58, 5.33, -26.33) mm, rotated rx -179.15 ry 0 rz -30.08 deg; joints [-3.356, -80.402, 141.264, -184.23, 60.737, 242.191]
  MoveC 4513 to (-316.6, 5.18, -26.33) mm, rotated rx -179.15 ry 0 rz -30.08 deg; joints [-3.358, -80.392, 141.267, -184.231, 60.75, 242.191] to (-316.66, 5.05, -26.33) mm, rotated rx -179.15 ry 0 rz -30.08 deg; joints [-3.361, -80.383, 141.27, -184.234, 60.762, 242.191]
  MoveL 4514 to (-316.66, 5.05, -26.33) mm, rotated rx -179.15 ry 0 rz -30.08 deg; joints [-3.361, -80.383, 141.27, -184.234, 60.762, 242.191]
  MoveL 4515 to (-327.16, -13.08, -26.33) mm, rotated rx -179.15 ry 0 rz -30.08 deg; joints [-3.948, -79.082, 141.603, -184.831, 62.413, 242.36]
  MoveC 4516 to (-327.25, -13.19, -26.33) mm, rotated rx -179.15 ry 0 rz -30.08 deg; joints [-3.953, -79.074, 141.605, -184.836, 62.424, 242.362] to (-327.36, -13.29, -26.33) mm, rotated rx -179.15 ry 0 rz -30.08 deg; joints [-3.959, -79.067, 141.606, -184.843, 62.432, 242.364]
  MoveL 4517 to (-327.36, -13.29, -26.33) mm, rotated rx -179.15 ry 0 rz -30.08 deg; joints [-3.959, -79.067, 141.606, -184.843, 62.432, 242.364]
  MoveC 4518 to (-327.47, -13.38, -26.33) mm, rotated rx -179.15 ry 0 rz -30.08 deg; joints [-3.965, -79.06, 141.608, -184.85, 62.441, 242.366] to (-327.55, -13.5, -26.33) mm, rotated rx -179.15 ry 0 rz -30.08 deg; joints [-3.97, -79.051, 141.61, -184.855, 62.451, 242.368]
  MoveL 4519 to (-327.55, -13.5, -26.33) mm, rotated rx -179.15 ry 0 rz -30.08 deg; joints [-3.97, -79.051, 141.61, -184.855, 62.451, 242.368]
  MoveC 4520 to (-328.23, -14.66, -26.88) mm, rotated rx -179.15 ry 0 rz -30.08 deg; joints [-4.006, -78.935, 141.59, -184.89, 62.549, 242.377] to (-328.51, -15.14, -28.23) mm, rotated rx -179.15 ry 0 rz -30.08 deg; joints [-4.016, -78.825, 141.501, -184.901, 62.57, 242.38]
  MoveL 4521 to (-328.51, -15.14, -28.23) mm, rotated rx -179.15 ry 0 rz -30.08 deg; joints [-4.016, -78.825, 141.501, -184.901, 62.57, 242.38]
  MoveL 4522 to (-328.51, -15.14, -30.77) mm, rotated rx -179.15 ry 0 rz -30.08 deg; joints [-4.006, -78.684, 141.318, -184.892, 62.529, 242.379]
  MoveC 4523 to (-328.23, -14.66, -32.12) mm, rotated rx -179.15 ry 0 rz -30.08 deg; joints [-3.986, -78.644, 141.213, -184.872, 62.463, 242.375] to (-327.55, -13.5, -32.67) mm, rotated rx -179.15 ry 0 rz -30.08 deg; joints [-3.946, -78.697, 141.153, -184.832, 62.348, 242.365]
  MoveL 4524 to (-327.55, -13.5, -32.67) mm, rotated rx -179.15 ry 0 rz -30.08 deg; joints [-3.946, -78.697, 141.153, -184.832, 62.348, 242.365]
  MoveC 4525 to (-327.47, -13.38, -32.67) mm, rotated rx -179.15 ry 0 rz -30.08 deg; joints [-3.941, -78.706, 141.151, -184.827, 62.338, 242.364] to (-327.36, -13.29, -32.67) mm, rotated rx -179.15 ry 0 rz -30.08 deg; joints [-3.935, -78.713, 141.15, -184.821, 62.329, 242.361]
  MoveL 4526 to (-327.36, -13.29, -32.67) mm, rotated rx -179.15 ry 0 rz -30.08 deg; joints [-3.935, -78.713, 141.15, -184.821, 62.329, 242.361]
  MoveC 4527 to (-327.25, -13.19, -32.67) mm, rotated rx -179.15 ry 0 rz -30.08 deg; joints [-3.929, -78.72, 141.149, -184.814, 62.321, 242.359] to (-327.16, -13.08, -32.67) mm, rotated rx -179.15 ry 0 rz -30.08 deg; joints [-3.924, -78.728, 141.147, -184.809, 62.31, 242.357]
  MoveL 4528 to (-327.16, -13.08, -32.67) mm, rotated rx -179.15 ry 0 rz -30.08 deg; joints [-3.924, -78.728, 141.147, -184.809, 62.31, 242.357]
  MoveL 4529 to (-316.66, 5.05, -32.67) mm, rotated rx -179.15 ry 0 rz -30.08 deg; joints [-3.341, -80.018, 140.816, -184.214, 60.673, 242.188]
  MoveC 4530 to (-316.6, 5.19, -32.67) mm, rotated rx -179.15 ry 0 rz -30.08 deg; joints [-3.337, -80.027, 140.813, -184.211, 60.661, 242.187] to (-316.58, 5.33, -32.67) mm, rotated rx -179.15 ry 0 rz -30.08 deg; joints [-3.336, -80.037, 140.81, -184.21, 60.648, 242.187]
  MoveL 4531 to (-316.58, 5.33, -32.67) mm, rotated rx -179.15 ry 0 rz -30.08 deg; joints [-3.336, -80.037, 140.81, -184.21, 60.648, 242.187]
  MoveC 4532 to (-316.55, 5.47, -32.67) mm, rotated rx -179.15 ry 0 rz -30.08 deg; joints [-3.335, -80.047, 140.807, -184.209, 60.635, 242.187] to (-316.49, 5.6, -32.67) mm, rotated rx -179.15 ry 0 rz -30.08 deg; joints [-3.331, -80.056, 140.804, -184.206, 60.623, 242.187]
  MoveL 4533 to (-316.49, 5.6, -32.67) mm, rotated rx -179.15 ry 0 rz -30.08 deg; joints [-3.331, -80.056, 140.804, -184.206, 60.623, 242.187]
  MoveC 4534 to (-315.82, 6.77, -33.23) mm, rotated rx -179.15 ry 0 rz -30.08 deg; joints [-3.292, -80.105, 140.742, -184.165, 60.51, 242.174] to (-315.54, 7.25, -34.58) mm, rotated rx -179.15 ry 0 rz -30.08 deg; joints [-3.272, -80.061, 140.636, -184.145, 60.447, 242.168]
  MoveL 4535 to (-315.54, 7.25, -34.58) mm, rotated rx -179.15 ry 0 rz -30.08 deg; joints [-3.272, -80.061, 140.636, -184.145, 60.447, 242.168]
  MoveL 4536 to (-315.54, 7.25, -37.12) mm, rotated rx -179.15 ry 0 rz -30.08 deg; joints [-3.264, -79.916, 140.454, -184.138, 60.411, 242.167]
  MoveC 4537 to (-315.82, 6.77, -38.47) mm, rotated rx -179.15 ry 0 rz -30.08 deg; joints [-3.276, -79.805, 140.367, -184.15, 60.435, 242.171] to (-316.49, 5.6, -39.02) mm, rotated rx -179.15 ry 0 rz -30.08 deg; joints [-3.311, -79.692, 140.349, -184.187, 60.531, 242.183]
  MoveL 4538 to (-316.49, 5.6, -39.02) mm, rotated rx -179.15 ry 0 rz -30.08 deg; joints [-3.311, -79.692, 140.349, -184.187, 60.531, 242.183]
  MoveC 4539 to (-316.55, 5.47, -39.02) mm, rotated rx -179.15 ry 0 rz -30.08 deg; joints [-3.315, -79.683, 140.352, -184.19, 60.543, 242.184] to (-316.58, 5.33, -39.02) mm, rotated rx -179.15 ry 0 rz -30.08 deg; joints [-3.316, -79.674, 140.355, -184.191, 60.556, 242.184]
  MoveL 4540 to (-316.58, 5.33, -39.02) mm, rotated rx -179.15 ry 0 rz -30.08 deg; joints [-3.316, -79.674, 140.355, -184.191, 60.556, 242.184]
  MoveC 4541 to (-316.6, 5.18, -39.02) mm, rotated rx -179.15 ry 0 rz -30.08 deg; joints [-3.317, -79.664, 140.358, -184.192, 60.568, 242.183] to (-316.66, 5.05, -39.02) mm, rotated rx -179.15 ry 0 rz -30.08 deg; joints [-3.321, -79.655, 140.361, -184.195, 60.58, 242.184]
  MoveL 4542 to (-316.66, 5.05, -39.02) mm, rotated rx -179.15 ry 0 rz -30.08 deg; joints [-3.321, -79.655, 140.361, -184.195, 60.58, 242.184]
  MoveL 4543 to (-327.16, -13.08, -39.02) mm, rotated rx -179.15 ry 0 rz -30.08 deg; joints [-3.901, -78.376, 140.689, -184.787, 62.204, 242.355]
  MoveC 4544 to (-327.25, -13.19, -39.02) mm, rotated rx -179.15 ry 0 rz -30.08 deg; joints [-3.905, -78.367, 140.691, -184.792, 62.215, 242.357] to (-327.36, -13.29, -39.02) mm, rotated rx -179.15 ry 0 rz -30.08 deg; joints [-3.912, -78.361, 140.692, -184.798, 62.223, 242.359]
  MoveL 4545 to (-327.36, -13.29, -39.02) mm, rotated rx -179.15 ry 0 rz -30.08 deg; joints [-3.912, -78.361, 140.692, -184.798, 62.223, 242.359]
  MoveC 4546 to (-327.47, -13.38, -39.02) mm, rotated rx -179.15 ry 0 rz -30.08 deg; joints [-3.918, -78.354, 140.694, -184.805, 62.232, 242.361] to (-327.55, -13.5, -39.02) mm, rotated rx -179.15 ry 0 rz -30.08 deg; joints [-3.922, -78.345, 140.696, -184.81, 62.242, 242.363]
  MoveL 4547 to (-327.55, -13.5, -39.02) mm, rotated rx -179.15 ry 0 rz -30.08 deg; joints [-3.922, -78.345, 140.696, -184.81, 62.242, 242.363]
  MoveC 4548 to (-328.23, -14.66, -39.58) mm, rotated rx -179.15 ry 0 rz -30.08 deg; joints [-3.958, -78.231, 140.675, -184.845, 62.337, 242.372] to (-328.51, -15.14, -40.93) mm, rotated rx -179.15 ry 0 rz -30.08 deg; joints [-3.968, -78.122, 140.586, -184.856, 62.357, 242.376]
  MoveL 4549 to (-328.51, -15.14, -40.93) mm, rotated rx -179.15 ry 0 rz -30.08 deg; joints [-3.968, -78.122, 140.586, -184.856, 62.357, 242.376]
  MoveL 4550 to (-328.51, -15.14, -43.47) mm, rotated rx -179.15 ry 0 rz -30.08 deg; joints [-3.959, -77.982, 140.402, -184.848, 62.313, 242.375]
  MoveC 4551 to (-328.23, -14.66, -44.81) mm, rotated rx -179.15 ry 0 rz -30.08 deg; joints [-3.938, -77.942, 140.297, -184.827, 62.247, 242.371] to (-327.55, -13.5, -45.37) mm, rotated rx -179.15 ry 0 rz -30.08 deg; joints [-3.899, -77.995, 140.237, -184.788, 62.133, 242.361]
  MoveL 4552 to (-327.55, -13.5, -45.37) mm, rotated rx -179.15 ry 0 rz -30.08 deg; joints [-3.899, -77.995, 140.237, -184.788, 62.133, 242.361]
  MoveC 4553 to (-327.47, -13.38, -45.37) mm, rotated rx -179.15 ry 0 rz -30.08 deg; joints [-3.894, -78.003, 140.235, -184.783, 62.123, 242.359] to (-327.36, -13.29, -45.37) mm, rotated rx -179.15 ry 0 rz -30.08 deg; joints [-3.888, -78.01, 140.234, -184.777, 62.115, 242.357]
  MoveL 4554 to (-327.36, -13.29, -45.37) mm, rotated rx -179.15 ry 0 rz -30.08 deg; joints [-3.888, -78.01, 140.234, -184.777, 62.115, 242.357]
  MoveC 4555 to (-327.25, -13.19, -45.37) mm, rotated rx -179.15 ry 0 rz -30.08 deg; joints [-3.882, -78.017, 140.232, -184.77, 62.106, 242.355] to (-327.16, -13.08, -45.37) mm, rotated rx -179.15 ry 0 rz -30.08 deg; joints [-3.877, -78.025, 140.231, -184.765, 62.096, 242.353]
  MoveL 4556 to (-327.16, -13.08, -45.37) mm, rotated rx -179.15 ry 0 rz -30.08 deg; joints [-3.877, -78.025, 140.231, -184.765, 62.096, 242.353]
  MoveL 4557 to (-316.66, 5.05, -45.37) mm, rotated rx -179.15 ry 0 rz -30.08 deg; joints [-3.301, -79.293, 139.904, -184.177, 60.485, 242.181]
  MoveC 4558 to (-316.6, 5.19, -45.37) mm, rotated rx -179.15 ry 0 rz -30.08 deg; joints [-3.298, -79.303, 139.902, -184.173, 60.473, 242.18] to (-316.58, 5.33, -45.37) mm, rotated rx -179.15 ry 0 rz -30.08 deg; joints [-3.296, -79.312, 139.899, -184.172, 60.46, 242.181]
  MoveL 4559 to (-316.58, 5.33, -45.37) mm, rotated rx -179.15 ry 0 rz -30.08 deg; joints [-3.296, -79.312, 139.899, -184.172, 60.46, 242.181]
  MoveC 4560 to (-316.55, 5.47, -45.37) mm, rotated rx -179.15 ry 0 rz -30.08 deg; joints [-3.295, -79.322, 139.896, -184.171, 60.448, 242.181] to (-316.49, 5.6, -45.37) mm, rotated rx -179.15 ry 0 rz -30.08 deg; joints [-3.292, -79.331, 139.893, -184.168, 60.436, 242.18]
  MoveL 4561 to (-316.49, 5.6, -45.37) mm, rotated rx -179.15 ry 0 rz -30.08 deg; joints [-3.292, -79.331, 139.893, -184.168, 60.436, 242.18]
  MoveC 4562 to (-315.82, 6.77, -45.93) mm, rotated rx -179.15 ry 0 rz -30.08 deg; joints [-3.253, -79.379, 139.83, -184.128, 60.324, 242.167] to (-315.54, 7.25, -47.28) mm, rotated rx -179.15 ry 0 rz -30.08 deg; joints [-3.233, -79.336, 139.724, -184.108, 60.261, 242.161]
  MoveL 4563 to (-315.54, 7.25, -47.28) mm, rotated rx -179.15 ry 0 rz -30.08 deg; joints [-3.233, -79.336, 139.724, -184.108, 60.261, 242.161]
  MoveL 4564 to (-315.54, 7.25, -49.82) mm, rotated rx -179.15 ry 0 rz -30.08 deg; joints [-3.226, -79.191, 139.541, -184.101, 60.222, 242.16]
  MoveC 4565 to (-315.82, 6.77, -51.16) mm, rotated rx -179.15 ry 0 rz -30.08 deg; joints [-3.237, -79.082, 139.454, -184.113, 60.244, 242.165] to (-316.49, 5.6, -51.72) mm, rotated rx -179.15 ry 0 rz -30.08 deg; joints [-3.272, -78.971, 139.436, -184.15, 60.338, 242.177]
  MoveL 4566 to (-316.49, 5.6, -51.72) mm, rotated rx -179.15 ry 0 rz -30.08 deg; joints [-3.272, -78.971, 139.436, -184.15, 60.338, 242.177]
  MoveC 4567 to (-316.55, 5.47, -51.72) mm, rotated rx -179.15 ry 0 rz -30.08 deg; joints [-3.275, -78.962, 139.438, -184.153, 60.35, 242.178] to (-316.58, 5.33, -51.72) mm, rotated rx -179.15 ry 0 rz -30.08 deg; joints [-3.277, -78.952, 139.441, -184.154, 60.362, 242.178]
  MoveL 4568 to (-316.58, 5.33, -51.72) mm, rotated rx -179.15 ry 0 rz -30.08 deg; joints [-3.277, -78.952, 139.441, -184.154, 60.362, 242.178]
  MoveC 4569 to (-316.6, 5.18, -51.72) mm, rotated rx -179.15 ry 0 rz -30.08 deg; joints [-3.278, -78.943, 139.444, -184.155, 60.375, 242.177] to (-316.66, 5.05, -51.72) mm, rotated rx -179.15 ry 0 rz -30.08 deg; joints [-3.281, -78.934, 139.447, -184.158, 60.386, 242.178]
  MoveL 4570 to (-316.66, 5.05, -51.72) mm, rotated rx -179.15 ry 0 rz -30.08 deg; joints [-3.281, -78.934, 139.447, -184.158, 60.386, 242.178]
  MoveL 4571 to (-327.16, -13.08, -51.72) mm, rotated rx -179.15 ry 0 rz -30.08 deg; joints [-3.854, -77.676, 139.771, -184.744, 61.985, 242.351]
  MoveC 4572 to (-327.25, -13.19, -51.72) mm, rotated rx -179.15 ry 0 rz -30.08 deg; joints [-3.859, -77.668, 139.773, -184.749, 61.995, 242.353] to (-327.36, -13.29, -51.72) mm, rotated rx -179.15 ry 0 rz -30.08 deg; joints [-3.865, -77.661, 139.774, -184.756, 62.003, 242.355]
  MoveL 4573 to (-327.36, -13.29, -51.72) mm, rotated rx -179.15 ry 0 rz -30.08 deg; joints [-3.865, -77.661, 139.774, -184.756, 62.003, 242.355]
  MoveC 4574 to (-327.47, -13.38, -51.72) mm, rotated rx -179.15 ry 0 rz -30.08 deg; joints [-3.871, -77.654, 139.775, -184.762, 62.012, 242.358] to (-327.55, -13.5, -51.72) mm, rotated rx -179.15 ry 0 rz -30.08 deg; joints [-3.876, -77.646, 139.777, -184.767, 62.022, 242.359]
  MoveL 4575 to (-327.55, -13.5, -51.72) mm, rotated rx -179.15 ry 0 rz -30.08 deg; joints [-3.876, -77.646, 139.777, -184.767, 62.022, 242.359]
  MoveC 4576 to (-328.23, -14.66, -52.28) mm, rotated rx -179.15 ry 0 rz -30.08 deg; joints [-3.911, -77.533, 139.756, -184.802, 62.115, 242.369] to (-328.51, -15.14, -53.63) mm, rotated rx -179.15 ry 0 rz -30.08 deg; joints [-3.921, -77.425, 139.666, -184.813, 62.133, 242.373]
  MoveL 4577 to (-328.51, -15.14, -53.63) mm, rotated rx -179.15 ry 0 rz -30.08 deg; joints [-3.921, -77.425, 139.666, -184.813, 62.133, 242.373]
  MoveL 4578 to (-328.51, -15.14, -56.16) mm, rotated rx -179.15 ry 0 rz -30.08 deg; joints [-3.912, -77.287, 139.482, -184.805, 62.087, 242.372]
  MoveC 4579 to (-328.23, -14.66, -57.51) mm, rotated rx -179.15 ry 0 rz -30.08 deg; joints [-3.892, -77.247, 139.376, -184.785, 62.02, 242.368] to (-327.55, -13.5, -58.07) mm, rotated rx -179.15 ry 0 rz -30.08 deg; joints [-3.853, -77.298, 139.316, -184.746, 61.908, 242.358]
  MoveL 4580 to (-327.55, -13.5, -58.07) mm, rotated rx -179.15 ry 0 rz -30.08 deg; joints [-3.853, -77.298, 139.316, -184.746, 61.908, 242.358]
  MoveC 4581 to (-327.47, -13.38, -58.07) mm, rotated rx -179.15 ry 0 rz -30.08 deg; joints [-3.848, -77.306, 139.314, -184.741, 61.898, 242.356] to (-327.36, -13.29, -58.07) mm, rotated rx -179.15 ry 0 rz -30.08 deg; joints [-3.842, -77.313, 139.313, -184.735, 61.889, 242.354]
  MoveL 4582 to (-327.36, -13.29, -58.07) mm, rotated rx -179.15 ry 0 rz -30.08 deg; joints [-3.842, -77.313, 139.313, -184.735, 61.889, 242.354]
  MoveC 4583 to (-327.25, -13.19, -58.07) mm, rotated rx -179.15 ry 0 rz -30.08 deg; joints [-3.836, -77.32, 139.311, -184.728, 61.881, 242.351] to (-327.16, -13.08, -58.07) mm, rotated rx -179.15 ry 0 rz -30.08 deg; joints [-3.832, -77.328, 139.31, -184.724, 61.871, 242.35]
  MoveL 4584 to (-327.16, -13.08, -58.07) mm, rotated rx -179.15 ry 0 rz -30.08 deg; joints [-3.832, -77.328, 139.31, -184.724, 61.871, 242.35]
  MoveL 4585 to (-316.66, 5.05, -58.07) mm, rotated rx -179.15 ry 0 rz -30.08 deg; joints [-3.262, -78.576, 138.988, -184.14, 60.285, 242.176]
  MoveC 4586 to (-316.6, 5.19, -58.07) mm, rotated rx -179.15 ry 0 rz -30.08 deg; joints [-3.259, -78.585, 138.985, -184.137, 60.273, 242.175] to (-316.58, 5.33, -58.07) mm, rotated rx -179.15 ry 0 rz -30.08 deg; joints [-3.258, -78.594, 138.982, -184.136, 60.261, 242.175]
  MoveL 4587 to (-316.58, 5.33, -58.07) mm, rotated rx -179.15 ry 0 rz -30.08 deg; joints [-3.258, -78.594, 138.982, -184.136, 60.261, 242.175]
  MoveC 4588 to (-316.55, 5.47, -58.07) mm, rotated rx -179.15 ry 0 rz -30.08 deg; joints [-3.256, -78.604, 138.979, -184.135, 60.249, 242.175] to (-316.49, 5.6, -58.07) mm, rotated rx -179.15 ry 0 rz -30.08 deg; joints [-3.253, -78.612, 138.977, -184.132, 60.237, 242.175]
  MoveL 4589 to (-316.49, 5.6, -58.07) mm, rotated rx -179.15 ry 0 rz -30.08 deg; joints [-3.253, -78.612, 138.977, -184.132, 60.237, 242.175]
  MoveC 4590 to (-315.82, 6.77, -58.63) mm, rotated rx -179.15 ry 0 rz -30.08 deg; joints [-3.215, -78.66, 138.914, -184.092, 60.126, 242.162] to (-315.54, 7.25, -59.97) mm, rotated rx -179.15 ry 0 rz -30.08 deg; joints [-3.196, -78.616, 138.808, -184.073, 60.062, 242.156]
  MoveL 4591 to (-315.54, 7.25, -59.97) mm, rotated rx -179.15 ry 0 rz -30.08 deg; joints [-3.196, -78.616, 138.808, -184.073, 60.062, 242.156]
  MoveL 4592 to (-315.54, 7.25, -62.51) mm, rotated rx -179.15 ry 0 rz -30.08 deg; joints [-3.188, -78.473, 138.624, -184.066, 60.021, 242.155]
  MoveC 4593 to (-315.82, 6.77, -63.86) mm, rotated rx -179.15 ry 0 rz -30.08 deg; joints [-3.199, -78.365, 138.535, -184.078, 60.042, 242.16] to (-316.49, 5.6, -64.42) mm, rotated rx -179.15 ry 0 rz -30.08 deg; joints [-3.234, -78.256, 138.517, -184.114, 60.134, 242.172]
  MoveL 4594 to (-316.49, 5.6, -64.42) mm, rotated rx -179.15 ry 0 rz -30.08 deg; joints [-3.234, -78.256, 138.517, -184.114, 60.134, 242.172]
  MoveC 4595 to (-316.55, 5.47, -64.42) mm, rotated rx -179.15 ry 0 rz -30.08 deg; joints [-3.237, -78.247, 138.52, -184.117, 60.145, 242.173] to (-316.58, 5.33, -64.42) mm, rotated rx -179.15 ry 0 rz -30.08 deg; joints [-3.239, -78.238, 138.522, -184.118, 60.157, 242.173]
  MoveL 4596 to (-316.58, 5.33, -64.42) mm, rotated rx -179.15 ry 0 rz -30.08 deg; joints [-3.239, -78.238, 138.522, -184.118, 60.157, 242.173]
  MoveC 4597 to (-316.6, 5.18, -64.42) mm, rotated rx -179.15 ry 0 rz -30.08 deg; joints [-3.24, -78.228, 138.525, -184.119, 60.17, 242.173] to (-316.66, 5.05, -64.42) mm, rotated rx -179.15 ry 0 rz -30.08 deg; joints [-3.243, -78.219, 138.528, -184.122, 60.181, 242.173]
  MoveL 4598 to (-316.66, 5.05, -64.42) mm, rotated rx -179.15 ry 0 rz -30.08 deg; joints [-3.243, -78.219, 138.528, -184.122, 60.181, 242.173]
  MoveL 4599 to (-327.16, -13.08, -64.42) mm, rotated rx -179.15 ry 0 rz -30.08 deg; joints [-3.809, -76.982, 138.847, -184.703, 61.755, 242.349]
  MoveC 4600 to (-327.25, -13.19, -64.42) mm, rotated rx -179.15 ry 0 rz -30.08 deg; joints [-3.814, -76.974, 138.849, -184.708, 61.765, 242.35] to (-327.36, -13.29, -64.42) mm, rotated rx -179.15 ry 0 rz -30.08 deg; joints [-3.82, -76.967, 138.851, -184.714, 61.773, 242.353]
  MoveL 4601 to (-327.36, -13.29, -64.42) mm, rotated rx -179.15 ry 0 rz -30.08 deg; joints [-3.82, -76.967, 138.851, -184.714, 61.773, 242.353]
  MoveC 4602 to (-327.47, -13.38, -64.42) mm, rotated rx -179.15 ry 0 rz -30.08 deg; joints [-3.826, -76.96, 138.852, -184.721, 61.781, 242.355] to (-327.55, -13.5, -64.42) mm, rotated rx -179.15 ry 0 rz -30.08 deg; joints [-3.83, -76.952, 138.854, -184.726, 61.791, 242.357]
  MoveL 4603 to (-327.55, -13.5, -64.42) mm, rotated rx -179.15 ry 0 rz -30.08 deg; joints [-3.83, -76.952, 138.854, -184.726, 61.791, 242.357]
  MoveC 4604 to (-328.23, -14.66, -64.98) mm, rotated rx -179.15 ry 0 rz -30.08 deg; joints [-3.865, -76.841, 138.832, -184.761, 61.882, 242.366] to (-328.51, -15.14, -66.32) mm, rotated rx -179.15 ry 0 rz -30.08 deg; joints [-3.875, -76.734, 138.742, -184.772, 61.898, 242.37]
  MoveL 4605 to (-328.51, -15.14, -66.32) mm, rotated rx -179.15 ry 0 rz -30.08 deg; joints [-3.875, -76.734, 138.742, -184.772, 61.898, 242.37]
  MoveL 4606 to (-328.51, -15.14, -68.86) mm, rotated rx -179.15 ry 0 rz -30.08 deg; joints [-3.866, -76.597, 138.556, -184.763, 61.85, 242.37]
  MoveC 4607 to (-328.23, -14.66, -70.21) mm, rotated rx -179.15 ry 0 rz -30.08 deg; joints [-3.846, -76.557, 138.45, -184.744, 61.783, 242.366] to (-327.55, -13.5, -70.77) mm, rotated rx -179.15 ry 0 rz -30.08 deg; joints [-3.808, -76.607, 138.39, -184.706, 61.672, 242.356]
  MoveL 4608 to (-327.55, -13.5, -70.77) mm, rotated rx -179.15 ry 0 rz -30.08 deg; joints [-3.808, -76.607, 138.39, -184.706, 61.672, 242.356]
  MoveC 4609 to (-327.47, -13.38, -70.77) mm, rotated rx -179.15 ry 0 rz -30.08 deg; joints [-3.803, -76.615, 138.388, -184.701, 61.662, 242.354] to (-327.36, -13.29, -70.77) mm, rotated rx -179.15 ry 0 rz -30.08 deg; joints [-3.798, -76.622, 138.387, -184.694, 61.654, 242.352]
  MoveL 4610 to (-327.36, -13.29, -70.77) mm, rotated rx -179.15 ry 0 rz -30.08 deg; joints [-3.798, -76.622, 138.387, -184.694, 61.654, 242.352]
  MoveC 4611 to (-327.25, -13.19, -70.77) mm, rotated rx -179.15 ry 0 rz -30.08 deg; joints [-3.792, -76.629, 138.386, -184.688, 61.646, 242.349] to (-327.16, -13.08, -70.77) mm, rotated rx -179.15 ry 0 rz -30.08 deg; joints [-3.787, -76.637, 138.384, -184.683, 61.636, 242.348]
  MoveL 4612 to (-327.16, -13.08, -70.77) mm, rotated rx -179.15 ry 0 rz -30.08 deg; joints [-3.787, -76.637, 138.384, -184.683, 61.636, 242.348]
  MoveL 4613 to (-316.66, 5.05, -70.77) mm, rotated rx -179.15 ry 0 rz -30.08 deg; joints [-3.224, -77.864, 138.067, -184.105, 60.074, 242.172]
  MoveC 4614 to (-316.6, 5.19, -70.77) mm, rotated rx -179.15 ry 0 rz -30.08 deg; joints [-3.221, -77.873, 138.064, -184.102, 60.063, 242.171] to (-316.58, 5.33, -70.77) mm, rotated rx -179.15 ry 0 rz -30.08 deg; joints [-3.22, -77.882, 138.061, -184.101, 60.051, 242.171]
  MoveL 4615 to (-316.58, 5.33, -70.77) mm, rotated rx -179.15 ry 0 rz -30.08 deg; joints [-3.22, -77.882, 138.061, -184.101, 60.051, 242.171]
  MoveC 4616 to (-316.55, 5.47, -70.77) mm, rotated rx -179.15 ry 0 rz -30.08 deg; joints [-3.218, -77.892, 138.058, -184.1, 60.039, 242.171] to (-316.49, 5.6, -70.77) mm, rotated rx -179.15 ry 0 rz -30.08 deg; joints [-3.215, -77.9, 138.056, -184.097, 60.027, 242.17]
  MoveL 4617 to (-316.49, 5.6, -70.77) mm, rotated rx -179.15 ry 0 rz -30.08 deg; joints [-3.215, -77.9, 138.056, -184.097, 60.027, 242.17]
  MoveC 4618 to (-315.82, 6.77, -71.32) mm, rotated rx -179.15 ry 0 rz -30.08 deg; joints [-3.177, -77.947, 137.993, -184.058, 59.917, 242.158] to (-315.54, 7.25, -72.67) mm, rotated rx -179.15 ry 0 rz -30.08 deg; joints [-3.159, -77.904, 137.886, -184.038, 59.853, 242.152]
  MoveL 4619 to (-315.54, 7.25, -72.67) mm, rotated rx -179.15 ry 0 rz -30.08 deg; joints [-3.159, -77.904, 137.886, -184.038, 59.853, 242.152]
  MoveL 4620 to (-315.54, 7.25, -75.21) mm, rotated rx -179.15 ry 0 rz -30.08 deg; joints [-3.151, -77.762, 137.702, -184.032, 59.81, 242.151]
